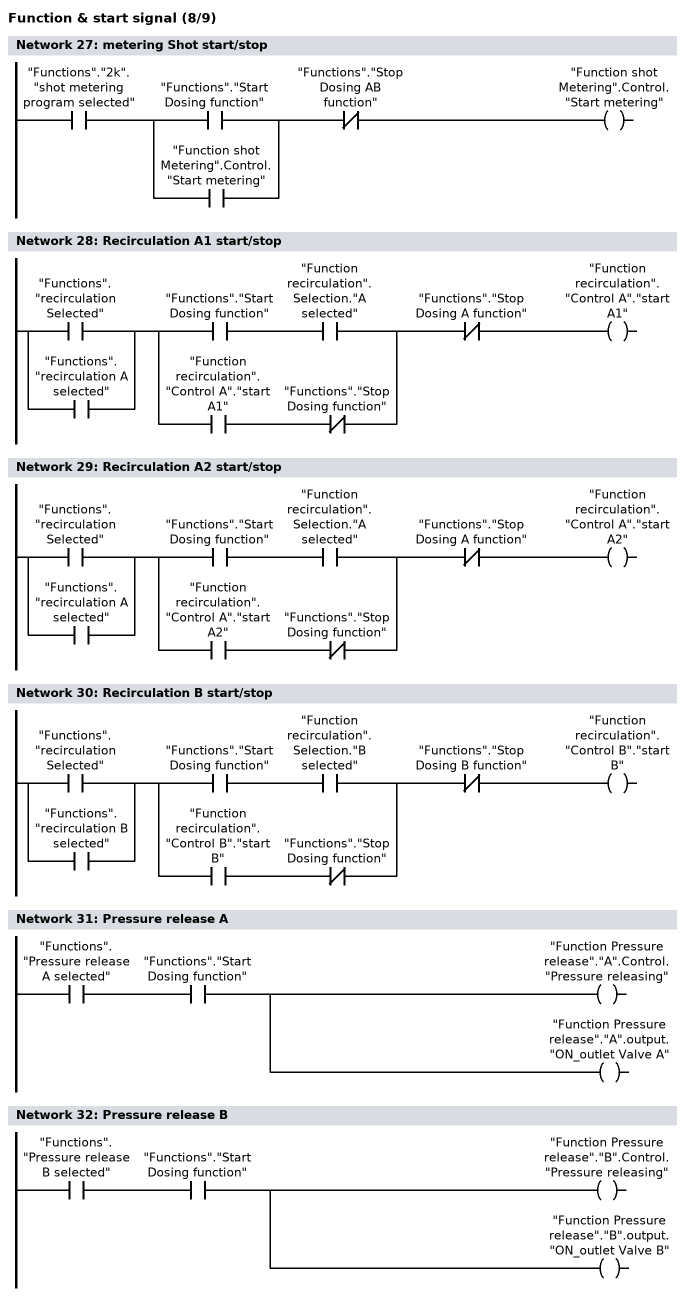
   RUNG wire#powerrail
      Contact( "Functions"."2k"."shot metering program selected" )
      wire#w1
      Contact( "Functions"."Start Dosing function" )
      wire#w2
      I_Contact( "Functions"."Stop Dosing AB function" )
      Coil( "Function shot Metering".Control."Start metering" )
   END_RUNG
   RUNG wire#w1
      Contact( "Function shot Metering".Control."Start metering" )
   END_RUNG wire#w2
   // the same network as SCL:
   "Function shot Metering".Control."Start metering" := "Functions"."2k"."shot metering program selected" AND ("Functions"."Start Dosing function" OR "Function shot Metering".Control."Start metering") AND NOT "Functions"."Stop Dosing AB function";
END_REGION

REGION Network 28: Recirculation A1 start/stop
   RUNG wire#powerrail
      Contact( "Functions"."recirculation Selected" )
      wire#w1
      Contact( "Functions"."Start Dosing function" )
      Contact( "Function recirculation".Selection."A selected" )
      wire#w2
      I_Contact( "Functions"."Stop Dosing A function" )
      Coil( "Function recirculation"."Control A"."start A1" )
   END_RUNG
   RUNG wire#powerrail
      Contact( "Functions"."recirculation A selected" )
   END_RUNG wire#w1
   RUNG wire#w1
      Contact( "Function recirculation"."Control A"."start A1" )
      I_Contact( "Functions"."Stop Dosing function" )
   END_RUNG wire#w2
   // the same network as SCL:
   "Function recirculation"."Control A"."start A1" := ("Functions"."recirculation Selected" OR "Functions"."recirculation A selected") AND (("Functions"."Start Dosing function" AND "Function recirculation".Selection."A selected") OR ("Function recirculation"."Control A"."start A1" AND NOT "Functions"."Stop Dosing function")) AND NOT "Functions"."Stop Dosing A function";
END_REGION

REGION Network 29: Recirculation A2 start/stop
   RUNG wire#powerrail
      Contact( "Functions"."recirculation Selected" )
      wire#w1
      Contact( "Functions"."Start Dosing function" )
      Contact( "Function recirculation".Selection."A selected" )
      wire#w2
      I_Contact( "Functions"."Stop Dosing A function" )
      Coil( "Function recirculation"."Control A"."start A2" )
   END_RUNG
   RUNG wire#powerrail
      Contact( "Functions"."recirculation A selected" )
   END_RUNG wire#w1
   RUNG wire#w1
      Contact( "Function recirculation"."Control A"."start A2" )
      I_Contact( "Functions"."Stop Dosing function" )
   END_RUNG wire#w2
   // the same network as SCL:
   "Function recirculation"."Control A"."start A2" := ("Functions"."recirculation Selected" OR "Functions"."recirculation A selected") AND (("Functions"."Start Dosing function" AND "Function recirculation".Selection."A selected") OR ("Function recirculation"."Control A"."start A2" AND NOT "Functions"."Stop Dosing function")) AND NOT "Functions"."Stop Dosing A function";
END_REGION

REGION Network 30: Recirculation B start/stop
   RUNG wire#powerrail
      Contact( "Functions"."recirculation Selected" )
      wire#w1
      Contact( "Functions"."Start Dosing function" )
      Contact( "Function recirculation".Selection."B selected" )
      wire#w2
      I_Contact( "Functions"."Stop Dosing B function" )
      Coil( "Function recirculation"."Control B"."start B" )
   END_RUNG
   RUNG wire#powerrail
      Contact( "Functions"."recirculation B selected" )
   END_RUNG wire#w1
   RUNG wire#w1
      Contact( "Function recirculation"."Control B"."start B" )
      I_Contact( "Functions"."Stop Dosing function" )
   END_RUNG wire#w2
   // the same network as SCL:
   "Function recirculation"."Control B"."start B" := ("Functions"."recirculation Selected" OR "Functions"."recirculation B selected") AND (("Functions"."Start Dosing function" AND "Function recirculation".Selection."B selected") OR ("Function recirculation"."Control B"."start B" AND NOT "Functions"."Stop Dosing function")) AND NOT "Functions"."Stop Dosing B function";
END_REGION

REGION Network 31: Pressure release A
   RUNG wire#powerrail
      Contact( "Functions"."Pressure release A selected" )
      Contact( "Functions"."Start Dosing function" )
      wire#w1
      Coil( "Function Pressure release"."A".Control."Pressure releasing" )
   END_RUNG
   RUNG wire#w1
      Coil( "Function Pressure release"."A".output."ON_outlet Valve A" )
   END_RUNG
   // the same network as SCL:
   "Function Pressure release"."A".Control."Pressure releasing" := "Functions"."Pressure release A selected" AND "Functions"."Start Dosing function";
   "Function Pressure release"."A".output."ON_outlet Valve A" := "Function Pressure release"."A".Control."Pressure releasing";
END_REGION

REGION Network 32: Pressure release B
   RUNG wire#powerrail
      Contact( "Functions"."Pressure release B selected" )
      Contact( "Functions"."Start Dosing function" )
      wire#w1
      Coil( "Function Pressure release"."B".Control."Pressure releasing" )
   END_RUNG
   RUNG wire#w1
      Coil( "Function Pressure release"."B".output."ON_outlet Valve B" )
   END_RUNG
   // the same network as SCL:
   "Function Pressure release"."B".Control."Pressure releasing" := "Functions"."Pressure release B selected" AND "Functions"."Start Dosing function";
   "Function Pressure release"."B".output."ON_outlet Valve B" := "Function Pressure release"."B".Control."Pressure releasing";
END_REGION

REGION Network 33: Pressure release AB
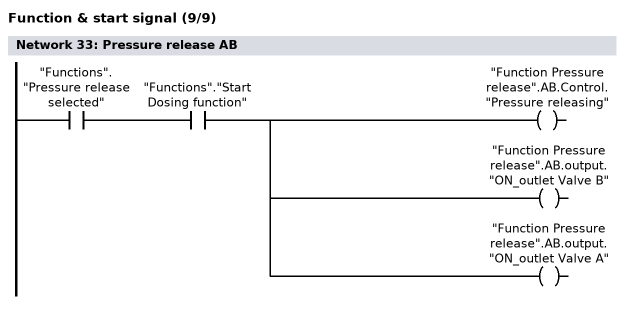
   RUNG wire#powerrail
      Contact( "Functions"."Pressure release selected" )
      Contact( "Functions"."Start Dosing function" )
      wire#w1
      Coil( "Function Pressure release".AB.Control."Pressure releasing" )
   END_RUNG
   RUNG wire#w1
      Coil( "Function Pressure release".AB.output."ON_outlet Valve B" )
   END_RUNG
   RUNG wire#w1
      Coil( "Function Pressure release".AB.output."ON_outlet Valve A" )
   END_RUNG
   // the same network as SCL:
   "Function Pressure release".AB.Control."Pressure releasing" := "Functions"."Pressure release selected" AND "Functions"."Start Dosing function";
   "Function Pressure release".AB.output."ON_outlet Valve B" := "Function Pressure release".AB.Control."Pressure releasing";
   "Function Pressure release".AB.output."ON_outlet Valve A" := "Function Pressure release".AB.Control."Pressure releasing";
END_REGION
END_FUNCTION

FUNCTION "Metering Program sequences" : Void   // FC2, LAD
{ S7_Optimized_Access := 'TRUE' }
VERSION : 0.1
// stored: AutoNumber true, IsIECCheckEnabled false, SetENOAutomatically false, UDAEnableTagReadback false
   VAR_TEMP
      temp1 : Bool;
   END_VAR
   VAR_TEMP   // added for the SCL form of the ladder/FBD networks
      _w1 : Bool;
   END_VAR
BEGIN

REGION Network 1: Do continous metering selection
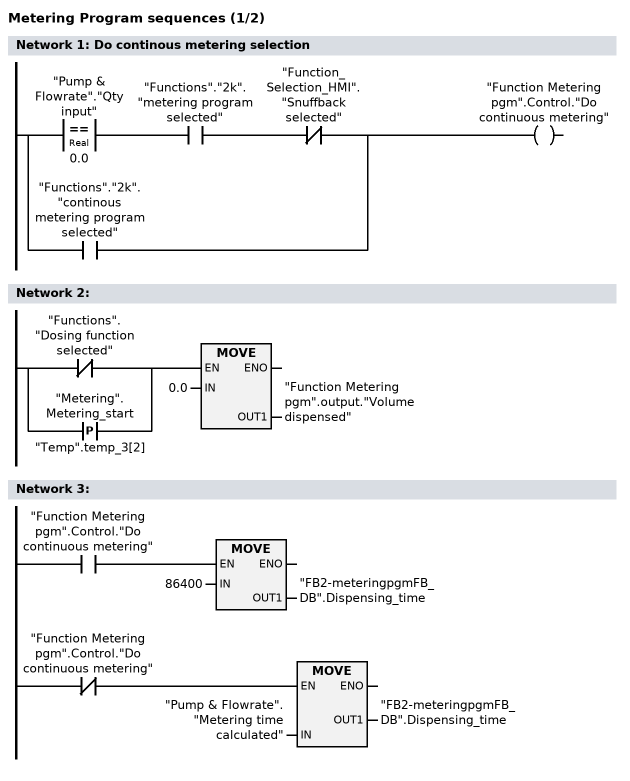
   RUNG wire#powerrail
      { S7_Templates := "SrcType := Real" } EQ_Contact(in1 := "Pump & Flowrate"."Qty input", in2 := 0.0)
      Contact( "Functions"."2k"."metering program selected" )
      I_Contact( "Function_Selection_HMI"."Snuffback selected" )
      wire#w1
      Coil( "Function Metering pgm".Control."Do continuous metering" )
   END_RUNG
   RUNG wire#powerrail
      Contact( "Functions"."2k"."continous metering program selected" )
   END_RUNG wire#w1
   // the same network as SCL:
   "Function Metering pgm".Control."Do continuous metering" := (("Pump & Flowrate"."Qty input" = 0.0) AND "Functions"."2k"."metering program selected" AND NOT "Function_Selection_HMI"."Snuffback selected") OR "Functions"."2k"."continous metering program selected";
END_REGION

REGION Network 2
   RUNG wire#powerrail
      I_Contact( "Functions"."Dosing function selected" )
      wire#w1
      Move(in := 0.0, out1 => "Function Metering pgm".output."Volume dispensed")
   END_RUNG
   RUNG wire#powerrail
      P_Contact(operand := "Metering".Metering_start, bit := "Temp".temp_3[2])
   END_RUNG wire#w1
   // the same network as SCL:
   #_w1 := "Metering".Metering_start AND NOT "Temp".temp_3[2];   // rising edge of "Metering".Metering_start
   "Temp".temp_3[2] := "Metering".Metering_start;
   IF NOT "Functions"."Dosing function selected" OR #_w1 THEN
       "Function Metering pgm".output."Volume dispensed" := 0.0;
   END_IF;
END_REGION

REGION Network 3
   RUNG wire#powerrail
      Contact( "Function Metering pgm".Control."Do continuous metering" )
      Move(in := 86400, out1 => "FB2-meteringpgmFB_DB".Dispensing_time)
   END_RUNG
   RUNG wire#powerrail
      I_Contact( "Function Metering pgm".Control."Do continuous metering" )
      Move(in := "Pump & Flowrate"."Metering time calculated", out1 => "FB2-meteringpgmFB_DB".Dispensing_time)
   END_RUNG
   // the same network as SCL:
   IF "Function Metering pgm".Control."Do continuous metering" THEN
       "FB2-meteringpgmFB_DB".Dispensing_time := 86400;
   END_IF;
   IF NOT "Function Metering pgm".Control."Do continuous metering" THEN
       "FB2-meteringpgmFB_DB".Dispensing_time := "Pump & Flowrate"."Metering time calculated";
   END_IF;
END_REGION

REGION Network 4
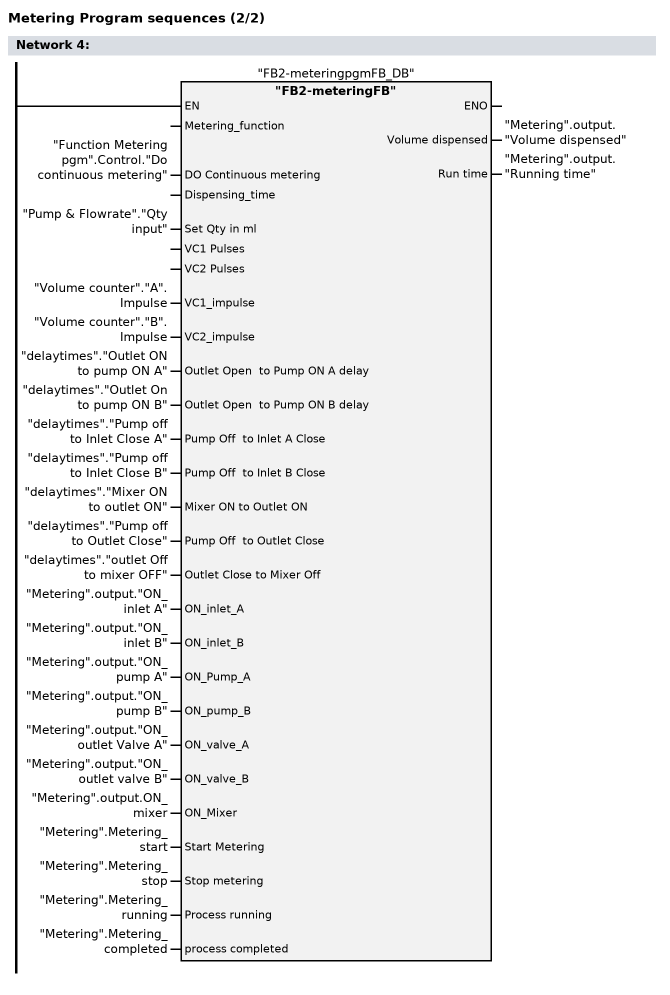
   RUNG wire#powerrail
      "FB2-meteringpgmFB_DB"(Metering_function :=, "DO Continuous metering" := "Function Metering pgm".Control."Do continuous metering", Dispensing_time :=, "Set Qty in ml" := "Pump & Flowrate"."Qty input", "VC1 Pulses" :=, "VC2 Pulses" :=, VC1_impulse := "Volume counter"."A".Impulse, VC2_impulse := "Volume counter"."B".Impulse, "Outlet Open  to Pump ON A delay" := "delaytimes"."Outlet ON to pump ON A", "Outlet Open  to Pump ON B delay" := "delaytimes"."Outlet On to pump ON B", "Pump Off  to Inlet A Close" := "delaytimes"."Pump off to Inlet Close A", "Pump Off  to Inlet B Close" := "delaytimes"."Pump off to Inlet Close B", "Mixer ON to Outlet ON" := "delaytimes"."Mixer ON to outlet ON", "Pump Off  to Outlet Close" := "delaytimes"."Pump off to Outlet Close", "Outlet Close to Mixer Off" := "delaytimes"."outlet Off to mixer OFF", ON_inlet_A := "Metering".output."ON_inlet A", ON_inlet_B := "Metering".output."ON_inlet B", ON_Pump_A := "Metering".output."ON_pump A", ON_pump_B := "Metering".output."ON_pump B", ON_valve_A := "Metering".output."ON_outlet Valve A", ON_valve_B := "Metering".output."ON_outlet valve B", ON_Mixer := "Metering".output.ON_mixer, "Start Metering" := "Metering".Metering_start, "Stop metering" := "Metering".Metering_stop, "Process running" := "Metering".Metering_running, "process completed" := "Metering".Metering_completed, "Volume dispensed" => "Metering".output."Volume dispensed", "Run time" => "Metering".output."Running time")
   END_RUNG
   // the same network as SCL:
   "FB2-meteringpgmFB_DB"("DO Continuous metering" := "Function Metering pgm".Control."Do continuous metering",   // "FB2-meteringFB"
                          "Set Qty in ml" := "Pump & Flowrate"."Qty input",
                          VC1_impulse := "Volume counter"."A".Impulse,
                          VC2_impulse := "Volume counter"."B".Impulse,
                          "Outlet Open  to Pump ON A delay" := "delaytimes"."Outlet ON to pump ON A",
                          "Outlet Open  to Pump ON B delay" := "delaytimes"."Outlet On to pump ON B",
                          "Pump Off  to Inlet A Close" := "delaytimes"."Pump off to Inlet Close A",
                          "Pump Off  to Inlet B Close" := "delaytimes"."Pump off to Inlet Close B",
                          "Mixer ON to Outlet ON" := "delaytimes"."Mixer ON to outlet ON",
                          "Pump Off  to Outlet Close" := "delaytimes"."Pump off to Outlet Close",
                          "Outlet Close to Mixer Off" := "delaytimes"."outlet Off to mixer OFF",
                          ON_inlet_A := "Metering".output."ON_inlet A",
                          ON_inlet_B := "Metering".output."ON_inlet B",
                          ON_Pump_A := "Metering".output."ON_pump A",
                          ON_pump_B := "Metering".output."ON_pump B",
                          ON_valve_A := "Metering".output."ON_outlet Valve A",
                          ON_valve_B := "Metering".output."ON_outlet valve B",
                          ON_Mixer := "Metering".output.ON_mixer,
                          "Start Metering" := "Metering".Metering_start,
                          "Stop metering" := "Metering".Metering_stop,
                          "Process running" := "Metering".Metering_running,
                          "process completed" := "Metering".Metering_completed,
                          "Volume dispensed" => "Metering".output."Volume dispensed",
                          "Run time" => "Metering".output."Running time");
END_REGION

REGION Network 5 (SCL)
   //IF NOT ("Gear Pump B On_REW") AND NOT ("Gear Pump A On_REW") THEN
       IF "Functions"."2k"."continous metering program selected" THEN
           "Function Continous Metering pgm".output."Volume dispensed" := "Metering".output."Volume dispensed";
           "Function Continous Metering pgm".output."Running time" := "Metering".output."Running time";
       ELSIF "Functions"."2k"."metering program selected" THEN
           "Function Metering pgm".output."Volume dispensed" := "Metering".output."Volume dispensed";
           "Function Metering pgm".output."Running time" := "Metering".output."Running time";
       ELSIF "Functions"."2k"."shot metering program selected" THEN
           "Function shot Metering".output."Volume dispensed" := "Metering".output."Volume dispensed";
           "Function shot Metering".output."Running time" := "Metering".output."Running time";
       ELSIF "Functions"."2k"."pre run program selected" THEN
           "Function Pre run".output."Volume dispensed" := "Metering".output."Volume dispensed";
           "Function Pre run".output."Running time" := "Metering".output."Running time";
       END_IF;
   //END_IF;
END_REGION

REGION Network 6 (SCL): Prerun Completed
   IF "Functions"."2k"."pre run program selected" AND "Metering".Metering_completed THEN //AND  ("Function Pre run".output."Volume dispensed" >="Pump & Flowrate"."Qty input")
       "Function Pre run".Control."metering completed" := TRUE;
   ELSIF "Function Flush"."Control A"."flush running" OR "Function Dearing with valve"."Control A"."dearing running"
       OR "Function Dearing with valve"."Control B"."dearing running" OR "Potlife".contol."Potlife elapsed machine not in regeneration"
           THEN //OR ("Functions"."2k"."pre run program selected"  AND "Functions"."Stop Dosing function")

       "Function Pre run".Control."metering completed" := FALSE;
   END_IF;
   "Control"."waiting For pre run" := NOT ("Function Pre run".Control."metering completed");
END_REGION
END_FUNCTION

FUNCTION_BLOCK "FB2-meteringFB"   // FB2, LAD
{ S7_Optimized_Access := 'TRUE' }
VERSION : 0.1
// stored: AutoNumber true, IsIECCheckEnabled false, IsRetainMemResEnabled false, MemoryReserve 100, SetENOAutomatically false, UDAEnableTagReadback false
   VAR_INPUT
      Metering_function : Int;
      "DO Continuous metering" : Bool;
      Dispensing_time : DInt;
      "Set Qty in ml" : Real;
      "VC1 Pulses" : DInt;
      "VC2 Pulses" : DInt;
      VC1_impulse : Real;
      VC2_impulse : Real;
      "Outlet Open  to Pump ON A delay" : DInt;
      "Outlet Open  to Pump ON B delay" : DInt;
      "Pump Off  to Inlet A Close" : DInt;
      "Pump Off  to Inlet B Close" : DInt;
      "Mixer ON to Outlet ON" : DInt;
      "Pump Off  to Outlet Close" : DInt;
      "Outlet Close to Mixer Off" : DInt;
   END_VAR
   VAR_OUTPUT
      "Volume dispensed" : Real;
      "Run time" : Int;
   END_VAR
   VAR_IN_OUT
      ON_inlet_A : Bool;
      ON_inlet_B : Bool;
      ON_Pump_A : Bool;
      ON_pump_B : Bool;
      ON_valve_A : Bool;
      ON_valve_B : Bool;
      ON_Mixer : Bool;
      "Start Metering" : Bool;
      "Stop metering" : Bool;
      "Process running" : Bool;
      "process completed" : Bool;
   END_VAR
   VAR
      "pump A to valveA delay" : Bool;
      "Pump B to valve B delay" : Bool;
      "Pump Off to mixer off delay_1" : Bool;
      "VC1 pulses prev" : DInt;
      "VC2 pulses prev" : DInt;
      "VC1 pulse generted" : DInt;
      "VC2 pulse generated" : DInt;
      "Pump A Voulme dispensed" : Real;
      "Pump B volume dispensed" : Real;
      "Total Volume dispensed" : Real;
      "metering started" : Bool;
      "metering time in msec" : DInt;
      "dispense time elapsed" : Bool;
      R_TRIG_Instance { S7_SetPoint := 'True'} : R_TRIG;
      IEC_Timer_0_Instance { S7_SetPoint := 'True'} : TON_TIME;
      IEC_Timer_0_Instance_1 { S7_SetPoint := 'True'} : TON_TIME;
      IEC_Timer_0_Instance_2 { S7_SetPoint := 'True'} : TON_TIME;
      R_TRIG_Instance_1 { S7_SetPoint := 'True'} : R_TRIG;
      temp { S7_SetPoint := 'True'} : Bool;
      IEC_Timer_0_Instance_3 { S7_SetPoint := 'True'} : TON_TIME;
      IEC_Timer_0_Instance_4 { S7_SetPoint := 'True'} : TON_TIME;
      IEC_Timer_0_Instance_5 { S7_SetPoint := 'True'} : TON_TIME;
      IEC_Timer_0_Instance_6 { S7_SetPoint := 'True'} : TON_TIME;
      IEC_Timer_0_Instance_7 { S7_SetPoint := 'True'} : TON_TIME;
      IEC_Timer_0_Instance_8 { S7_SetPoint := 'True'} : TON_TIME;
   END_VAR
   VAR_TEMP
      Ons_temp : Bool;
   END_VAR
   VAR_TEMP   // added for the SCL form of the ladder/FBD networks
      _w1 : Bool;
      _w2 : Bool;
      _w3 : Bool;
   END_VAR
BEGIN

REGION Network 1
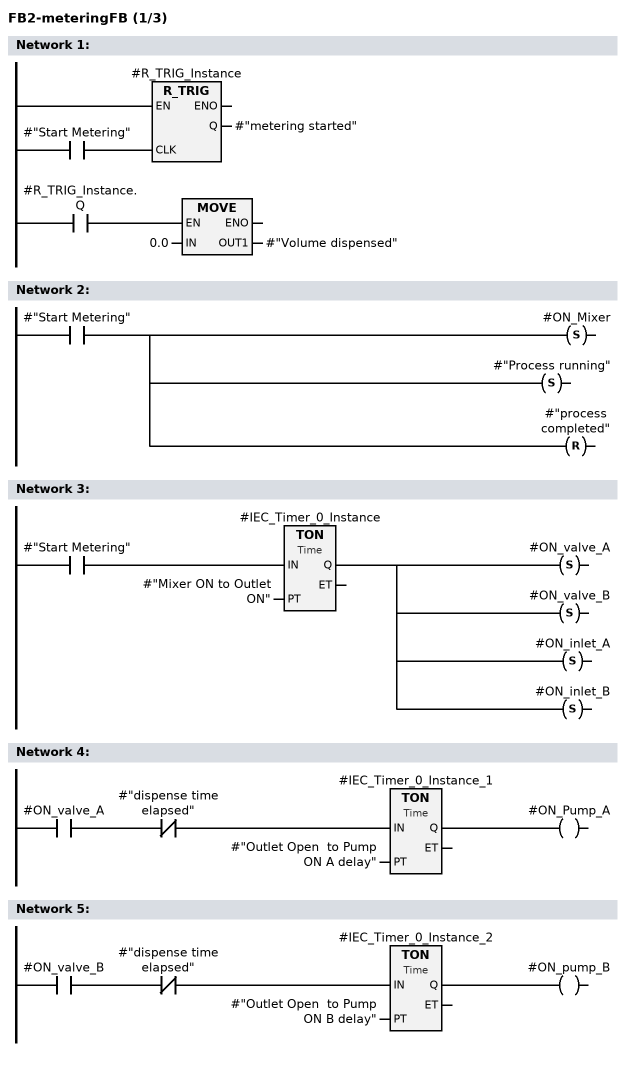
   RUNG wire#powerrail
      #R_TRIG_Instance.R_TRIG(CLK := wire#w1, Q => #"metering started")
   END_RUNG
   RUNG wire#powerrail
      Contact( #"Start Metering" )
   END_RUNG wire#w1
   RUNG wire#powerrail
      Contact( #R_TRIG_Instance.Q )
      Move(in := 0.0, out1 => #"Volume dispensed")
   END_RUNG
   // the same network as SCL:
   #R_TRIG_Instance(CLK := #"Start Metering", Q => #"metering started");   // R_TRIG
   IF #R_TRIG_Instance.Q THEN #"Volume dispensed" := 0.0; END_IF;
END_REGION

REGION Network 2
   RUNG wire#powerrail
      Contact( #"Start Metering" )
      wire#w1
      S_Coil( #ON_Mixer )
   END_RUNG
   RUNG wire#w1
      S_Coil( #"Process running" )
   END_RUNG
   RUNG wire#w1
      R_Coil( #"process completed" )
   END_RUNG
   // the same network as SCL:
   IF #"Start Metering" THEN
       #ON_Mixer := TRUE;
       #"Process running" := TRUE;
       #"process completed" := FALSE;
   END_IF;
END_REGION

REGION Network 3
   RUNG wire#powerrail
      Contact( #"Start Metering" )
      { S7_Templates := "time_type := Time" } #IEC_Timer_0_Instance.TON(pt := #"Mixer ON to Outlet ON", et =>)
      wire#w1
      S_Coil( #ON_valve_A )
   END_RUNG
   RUNG wire#w1
      S_Coil( #ON_valve_B )
   END_RUNG
   RUNG wire#w1
      S_Coil( #ON_inlet_A )
   END_RUNG
   RUNG wire#w1
      S_Coil( #ON_inlet_B )
   END_RUNG
   // the same network as SCL:
   #IEC_Timer_0_Instance(IN := #"Start Metering", PT := #"Mixer ON to Outlet ON");   // TON
   IF #IEC_Timer_0_Instance.Q THEN
       #ON_valve_A := TRUE;
       #ON_valve_B := TRUE;
       #ON_inlet_A := TRUE;
       #ON_inlet_B := TRUE;
   END_IF;
END_REGION

REGION Network 4
   RUNG wire#powerrail
      Contact( #ON_valve_A )
      I_Contact( #"dispense time elapsed" )
      { S7_Templates := "time_type := Time" } #IEC_Timer_0_Instance_1.TON(pt := #"Outlet Open  to Pump ON A delay", et =>)
      Coil( #ON_Pump_A )
   END_RUNG
   // the same network as SCL:
   #IEC_Timer_0_Instance_1(IN := #ON_valve_A AND NOT #"dispense time elapsed",   // TON
                           PT := #"Outlet Open  to Pump ON A delay");
   #ON_Pump_A := #IEC_Timer_0_Instance_1.Q;
END_REGION

REGION Network 5
   RUNG wire#powerrail
      Contact( #ON_valve_B )
      I_Contact( #"dispense time elapsed" )
      { S7_Templates := "time_type := Time" } #IEC_Timer_0_Instance_2.TON(pt := #"Outlet Open  to Pump ON B delay", et =>)
      Coil( #ON_pump_B )
   END_RUNG
   // the same network as SCL:
   #IEC_Timer_0_Instance_2(IN := #ON_valve_B AND NOT #"dispense time elapsed",   // TON
                           PT := #"Outlet Open  to Pump ON B delay");
   #ON_pump_B := #IEC_Timer_0_Instance_2.Q;
END_REGION

REGION Network 6
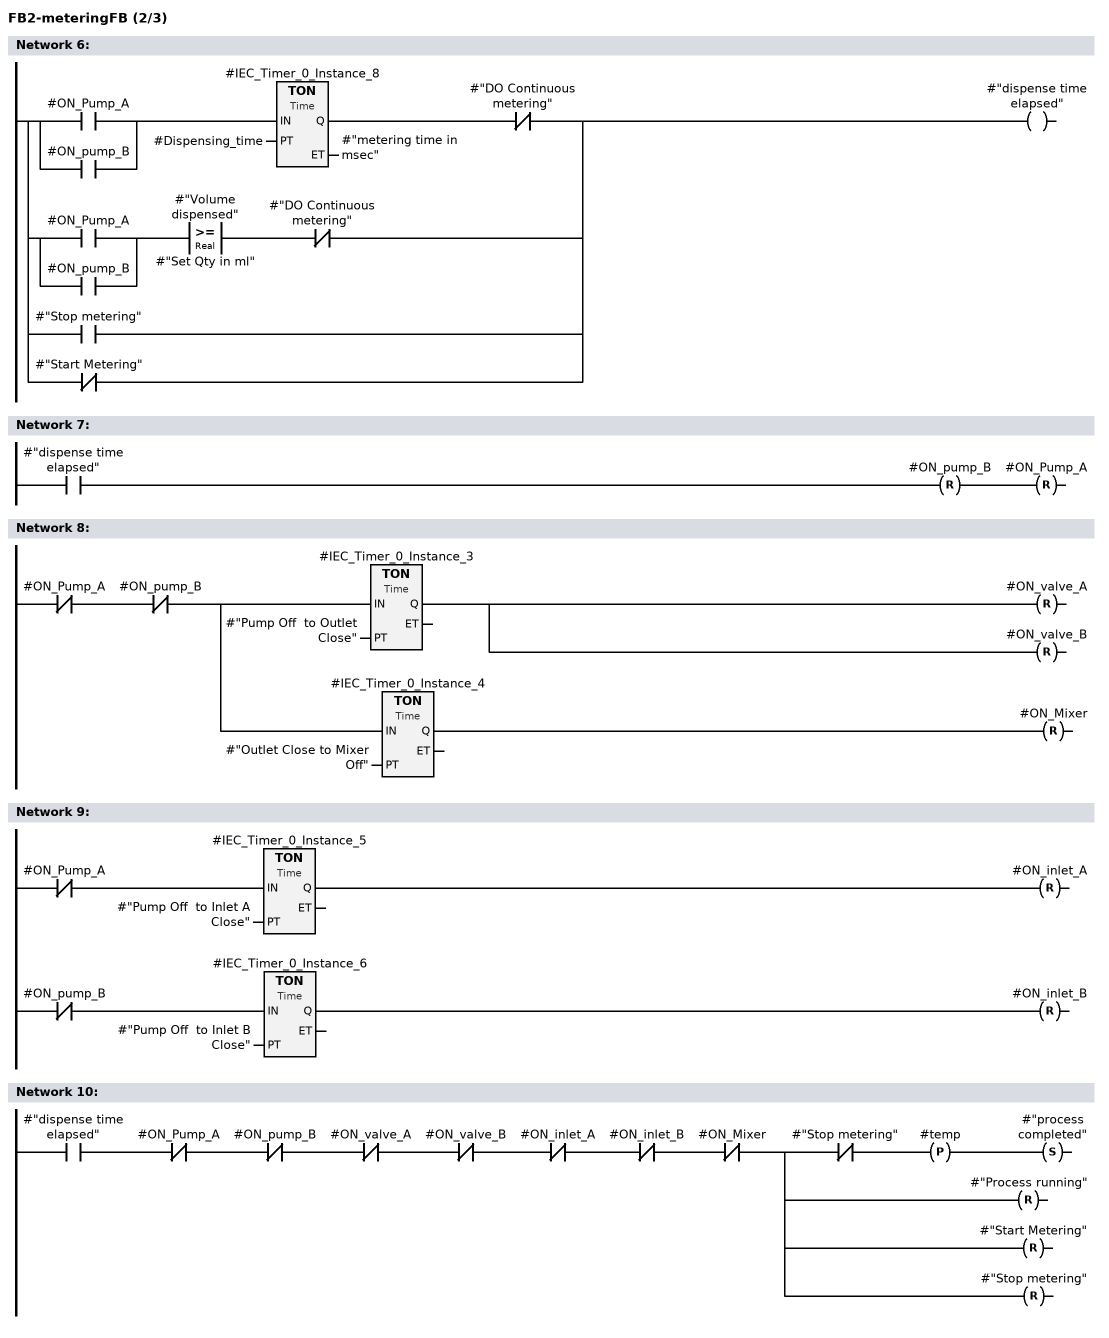
   RUNG wire#powerrail
      Contact( #ON_Pump_A )
      wire#w1
      { S7_Templates := "time_type := Time" } #IEC_Timer_0_Instance_8.TON(pt := #Dispensing_time, et => #"metering time in msec")
      I_Contact( #"DO Continuous metering" )
      wire#w2
      Coil( #"dispense time elapsed" )
   END_RUNG
   RUNG wire#powerrail
      Contact( #ON_pump_B )
   END_RUNG wire#w1
   RUNG wire#powerrail
      Contact( #ON_Pump_A )
      wire#w3
      { S7_Templates := "SrcType := Real" } GE_Contact(in1 := #"Volume dispensed", in2 := #"Set Qty in ml")
      I_Contact( #"DO Continuous metering" )
   END_RUNG wire#w2
   RUNG wire#powerrail
      Contact( #ON_pump_B )
   END_RUNG wire#w3
   RUNG wire#powerrail
      Contact( #"Stop metering" )
   END_RUNG wire#w2
   RUNG wire#powerrail
      I_Contact( #"Start Metering" )
   END_RUNG wire#w2
   // the same network as SCL:
   #IEC_Timer_0_Instance_8(IN := #ON_Pump_A OR #ON_pump_B,   // TON
                           PT := #Dispensing_time,
                           ET => #"metering time in msec");
   #"dispense time elapsed" := (#IEC_Timer_0_Instance_8.Q AND NOT #"DO Continuous metering") OR ((#ON_Pump_A OR #ON_pump_B) AND (#"Volume dispensed" >= #"Set Qty in ml") AND NOT #"DO Continuous metering") OR #"Stop metering" OR NOT #"Start Metering";
END_REGION

REGION Network 7
   RUNG wire#powerrail
      Contact( #"dispense time elapsed" )
      R_Coil( #ON_pump_B )
      R_Coil( #ON_Pump_A )
   END_RUNG
   // the same network as SCL:
   IF #"dispense time elapsed" THEN
       #ON_pump_B := FALSE;
       #ON_Pump_A := FALSE;
   END_IF;
END_REGION

REGION Network 8
   RUNG wire#powerrail
      I_Contact( #ON_Pump_A )
      I_Contact( #ON_pump_B )
      wire#w1
      { S7_Templates := "time_type := Time" } #IEC_Timer_0_Instance_3.TON(pt := #"Pump Off  to Outlet Close", et =>)
      wire#w2
      R_Coil( #ON_valve_A )
   END_RUNG
   RUNG wire#w2
      R_Coil( #ON_valve_B )
   END_RUNG
   RUNG wire#w1
      { S7_Templates := "time_type := Time" } #IEC_Timer_0_Instance_4.TON(pt := #"Outlet Close to Mixer Off", et =>)
      R_Coil( #ON_Mixer )
   END_RUNG
   // the same network as SCL:
   #_w1 := NOT #ON_Pump_A AND NOT #ON_pump_B;
   #IEC_Timer_0_Instance_3(IN := #_w1, PT := #"Pump Off  to Outlet Close");   // TON
   IF #IEC_Timer_0_Instance_3.Q THEN
       #ON_valve_A := FALSE;
       #ON_valve_B := FALSE;
   END_IF;
   #IEC_Timer_0_Instance_4(IN := #_w1, PT := #"Outlet Close to Mixer Off");   // TON
   IF #IEC_Timer_0_Instance_4.Q THEN #ON_Mixer := FALSE; END_IF;
END_REGION

REGION Network 9
   RUNG wire#powerrail
      I_Contact( #ON_Pump_A )
      { S7_Templates := "time_type := Time" } #IEC_Timer_0_Instance_5.TON(pt := #"Pump Off  to Inlet A Close", et =>)
      R_Coil( #ON_inlet_A )
   END_RUNG
   RUNG wire#powerrail
      I_Contact( #ON_pump_B )
      { S7_Templates := "time_type := Time" } #IEC_Timer_0_Instance_6.TON(pt := #"Pump Off  to Inlet B Close", et =>)
      R_Coil( #ON_inlet_B )
   END_RUNG
   // the same network as SCL:
   #IEC_Timer_0_Instance_5(IN := NOT #ON_Pump_A, PT := #"Pump Off  to Inlet A Close");   // TON
   IF #IEC_Timer_0_Instance_5.Q THEN #ON_inlet_A := FALSE; END_IF;
   #IEC_Timer_0_Instance_6(IN := NOT #ON_pump_B, PT := #"Pump Off  to Inlet B Close");   // TON
   IF #IEC_Timer_0_Instance_6.Q THEN #ON_inlet_B := FALSE; END_IF;
END_REGION

REGION Network 10
   RUNG wire#powerrail
      Contact( #"dispense time elapsed" )
      I_Contact( #ON_Pump_A )
      I_Contact( #ON_pump_B )
      I_Contact( #ON_valve_A )
      I_Contact( #ON_valve_B )
      I_Contact( #ON_inlet_A )
      I_Contact( #ON_inlet_B )
      I_Contact( #ON_Mixer )
      wire#w1
      I_Contact( #"Stop metering" )
      P_Trig( #temp )
      S_Coil( #"process completed" )
   END_RUNG
   RUNG wire#w1
      R_Coil( #"Process running" )
   END_RUNG
   RUNG wire#w1
      R_Coil( #"Start Metering" )
   END_RUNG
   RUNG wire#w1
      R_Coil( #"Stop metering" )
   END_RUNG
   // the same network as SCL:
   #_w1 := #"dispense time elapsed" AND NOT #ON_Pump_A AND NOT #ON_pump_B AND NOT #ON_valve_A AND NOT #ON_valve_B AND NOT #ON_inlet_A AND NOT #ON_inlet_B AND NOT #ON_Mixer;
   #_w2 := #_w1 AND NOT #"Stop metering";
   #_w3 := #_w2 AND NOT #temp;   // rising edge
   #temp := #_w2;
   IF #_w3 THEN #"process completed" := TRUE; END_IF;
   IF #_w1 THEN
       #"Process running" := FALSE;
       #"Start Metering" := FALSE;
       #"Stop metering" := FALSE;
   END_IF;
END_REGION

REGION Network 11
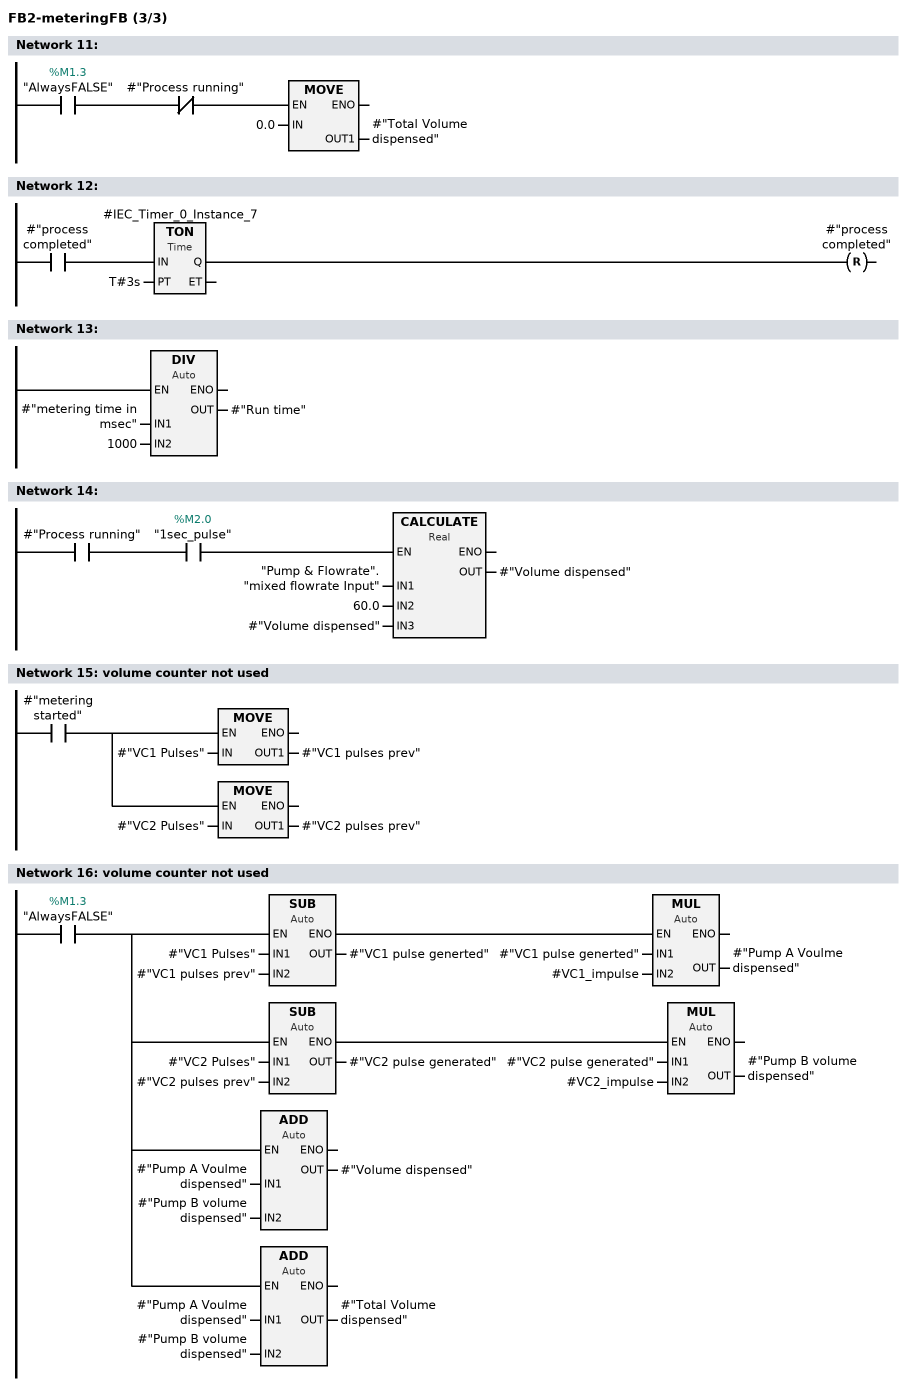
   RUNG wire#powerrail
      Contact( "AlwaysFALSE" )
      I_Contact( #"Process running" )
      Move(in := 0.0, out1 => #"Total Volume dispensed")
   END_RUNG
   // the same network as SCL:
   IF "AlwaysFALSE" AND NOT #"Process running" THEN #"Total Volume dispensed" := 0.0; END_IF;
END_REGION

REGION Network 12
   RUNG wire#powerrail
      Contact( #"process completed" )
      { S7_Templates := "time_type := Time" } #IEC_Timer_0_Instance_7.TON(pt := T#3s, et =>)
      R_Coil( #"process completed" )
   END_RUNG
   // the same network as SCL:
   #IEC_Timer_0_Instance_7(IN := #"process completed", PT := T#3s);   // TON
   IF #IEC_Timer_0_Instance_7.Q THEN #"process completed" := FALSE; END_IF;
END_REGION

REGION Network 13
   RUNG wire#powerrail
      Div(in1 := #"metering time in msec", in2 := 1000, out => #"Run time")
   END_RUNG
   // the same network as SCL:
   #"Run time" := #"metering time in msec" / 1000;
END_REGION

REGION Network 14
   RUNG wire#powerrail
      Contact( #"Process running" )
      Contact( "1sec_pulse" )
      { S7_Templates := "SrcType := Real"; S7_Expression := "(IN1/IN2)+IN3" } Calculate(in1 := "Pump & Flowrate"."mixed flowrate Input", in2 := 60.0, in3 := #"Volume dispensed", out => #"Volume dispensed")
   END_RUNG
   // the same network as SCL:
   IF #"Process running" AND "1sec_pulse" THEN
       #"Volume dispensed" := ("Pump & Flowrate"."mixed flowrate Input"/60.0)+#"Volume dispensed";
   END_IF;
END_REGION

REGION Network 15: volume counter not used
   RUNG wire#powerrail
      Contact( #"metering started" )
      wire#w1
      Move(in := #"VC1 Pulses", out1 => #"VC1 pulses prev")
   END_RUNG
   RUNG wire#w1
      Move(in := #"VC2 Pulses", out1 => #"VC2 pulses prev")
   END_RUNG
   // the same network as SCL:
   IF #"metering started" THEN
       #"VC1 pulses prev" := #"VC1 Pulses";
       #"VC2 pulses prev" := #"VC2 Pulses";
   END_IF;
END_REGION

REGION Network 16: volume counter not used
   RUNG wire#powerrail
      Contact( "AlwaysFALSE" )
      wire#w1
      Sub(in1 := #"VC1 Pulses", in2 := #"VC1 pulses prev", out => #"VC1 pulse generted")
      Mul(in1 := #"VC1 pulse generted", in2 := #VC1_impulse, out => #"Pump A Voulme dispensed")
   END_RUNG
   RUNG wire#w1
      Sub(in1 := #"VC2 Pulses", in2 := #"VC2 pulses prev", out => #"VC2 pulse generated")
      Mul(in1 := #"VC2 pulse generated", in2 := #VC2_impulse, out => #"Pump B volume dispensed")
   END_RUNG
   RUNG wire#w1
      Add(in1 := #"Pump A Voulme dispensed", in2 := #"Pump B volume dispensed", out => #"Volume dispensed")
   END_RUNG
   RUNG wire#w1
      Add(in1 := #"Pump A Voulme dispensed", in2 := #"Pump B volume dispensed", out => #"Total Volume dispensed")
   END_RUNG
   // the same network as SCL:
   IF "AlwaysFALSE" THEN
       #"VC1 pulse generted" := #"VC1 Pulses" - #"VC1 pulses prev";
       #"Pump A Voulme dispensed" := #"VC1 pulse generted" * #VC1_impulse;
       #"VC2 pulse generated" := #"VC2 Pulses" - #"VC2 pulses prev";
       #"Pump B volume dispensed" := #"VC2 pulse generated" * #VC2_impulse;
       #"Volume dispensed" := #"Pump A Voulme dispensed" + #"Pump B volume dispensed";
       #"Total Volume dispensed" := #"Pump A Voulme dispensed" + #"Pump B volume dispensed";
   END_IF;
END_REGION
END_FUNCTION_BLOCK

FUNCTION "Ratio Check Program sequences" : Void   // FC6, LAD
{ S7_Optimized_Access := 'TRUE' }
VERSION : 0.1
// stored: AutoNumber true, IsIECCheckEnabled false, SetENOAutomatically false, UDAEnableTagReadback false
   VAR_TEMP
      temp1 : Bool;
   END_VAR
   VAR_TEMP   // added for the SCL form of the ladder/FBD networks
      _w1 : Bool;
      _w2 : Bool;
      _w3 : Bool;
      _w4 : Bool;
   END_VAR
BEGIN

REGION Network 1
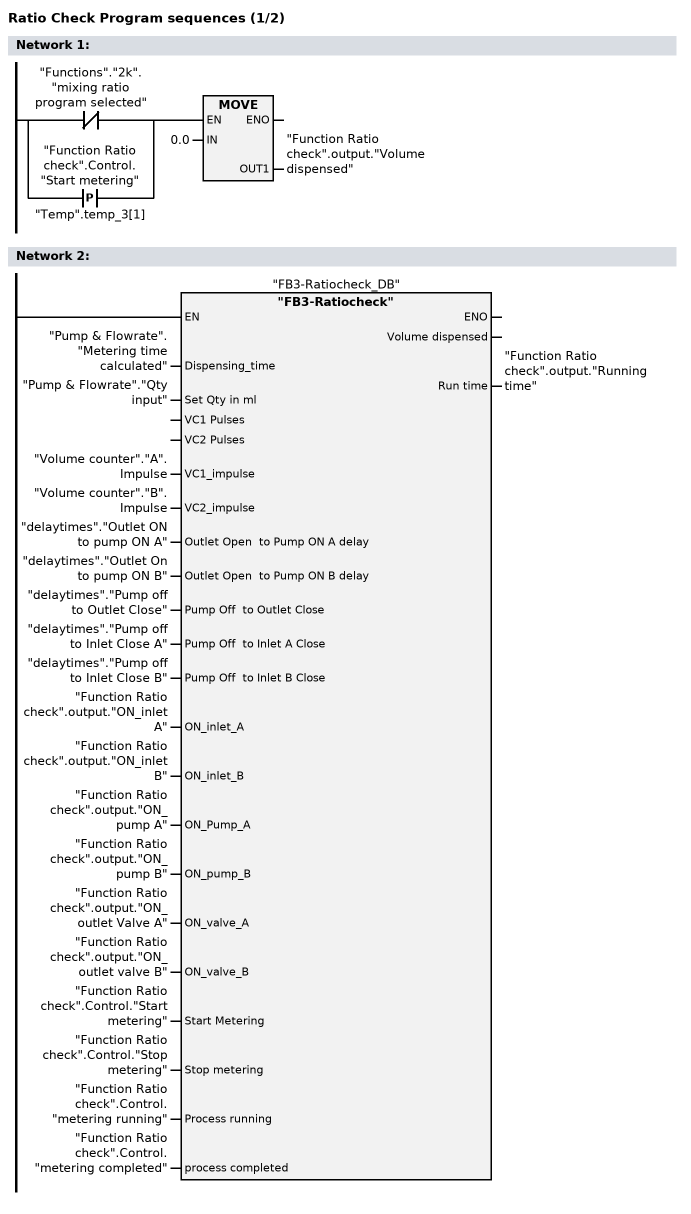
   RUNG wire#powerrail
      I_Contact( "Functions"."2k"."mixing ratio program selected" )
      wire#w1
      Move(in := 0.0, out1 => "Function Ratio check".output."Volume dispensed")
   END_RUNG
   RUNG wire#powerrail
      P_Contact(operand := "Function Ratio check".Control."Start metering", bit := "Temp".temp_3[1])
   END_RUNG wire#w1
   // the same network as SCL:
   #_w1 := "Function Ratio check".Control."Start metering" AND NOT "Temp".temp_3[1];   // rising edge of "Function Ratio check".Control."Start metering"
   "Temp".temp_3[1] := "Function Ratio check".Control."Start metering";
   IF NOT "Functions"."2k"."mixing ratio program selected" OR #_w1 THEN
       "Function Ratio check".output."Volume dispensed" := 0.0;
   END_IF;
END_REGION

REGION Network 2
   RUNG wire#powerrail
      "FB3-Ratiocheck_DB"(Dispensing_time := "Pump & Flowrate"."Metering time calculated", "Set Qty in ml" := "Pump & Flowrate"."Qty input", "VC1 Pulses" :=, "VC2 Pulses" :=, VC1_impulse := "Volume counter"."A".Impulse, VC2_impulse := "Volume counter"."B".Impulse, "Outlet Open  to Pump ON A delay" := "delaytimes"."Outlet ON to pump ON A", "Outlet Open  to Pump ON B delay" := "delaytimes"."Outlet On to pump ON B", "Pump Off  to Outlet Close" := "delaytimes"."Pump off to Outlet Close", "Pump Off  to Inlet A Close" := "delaytimes"."Pump off to Inlet Close A", "Pump Off  to Inlet B Close" := "delaytimes"."Pump off to Inlet Close B", ON_inlet_A := "Function Ratio check".output."ON_inlet A", ON_inlet_B := "Function Ratio check".output."ON_inlet B", ON_Pump_A := "Function Ratio check".output."ON_pump A", ON_pump_B := "Function Ratio check".output."ON_pump B", ON_valve_A := "Function Ratio check".output."ON_outlet Valve A", ON_valve_B := "Function Ratio check".output."ON_outlet valve B", "Start Metering" := "Function Ratio check".Control."Start metering", "Stop metering" := "Function Ratio check".Control."Stop metering", "Process running" := "Function Ratio check".Control."metering running", "process completed" := "Function Ratio check".Control."metering completed", "Volume dispensed" =>, "Run time" => "Function Ratio check".output."Running time")
   END_RUNG
   // the same network as SCL:
   "FB3-Ratiocheck_DB"(Dispensing_time := "Pump & Flowrate"."Metering time calculated",   // "FB3-Ratiocheck"
                       "Set Qty in ml" := "Pump & Flowrate"."Qty input",
                       VC1_impulse := "Volume counter"."A".Impulse,
                       VC2_impulse := "Volume counter"."B".Impulse,
                       "Outlet Open  to Pump ON A delay" := "delaytimes"."Outlet ON to pump ON A",
                       "Outlet Open  to Pump ON B delay" := "delaytimes"."Outlet On to pump ON B",
                       "Pump Off  to Outlet Close" := "delaytimes"."Pump off to Outlet Close",
                       "Pump Off  to Inlet A Close" := "delaytimes"."Pump off to Inlet Close A",
                       "Pump Off  to Inlet B Close" := "delaytimes"."Pump off to Inlet Close B",
                       ON_inlet_A := "Function Ratio check".output."ON_inlet A",
                       ON_inlet_B := "Function Ratio check".output."ON_inlet B",
                       ON_Pump_A := "Function Ratio check".output."ON_pump A",
                       ON_pump_B := "Function Ratio check".output."ON_pump B",
                       ON_valve_A := "Function Ratio check".output."ON_outlet Valve A",
                       ON_valve_B := "Function Ratio check".output."ON_outlet valve B",
                       "Start Metering" := "Function Ratio check".Control."Start metering",
                       "Stop metering" := "Function Ratio check".Control."Stop metering",
                       "Process running" := "Function Ratio check".Control."metering running",
                       "process completed" := "Function Ratio check".Control."metering completed",
                       "Run time" => "Function Ratio check".output."Running time");
END_REGION

REGION Network 3: Volume dispensed
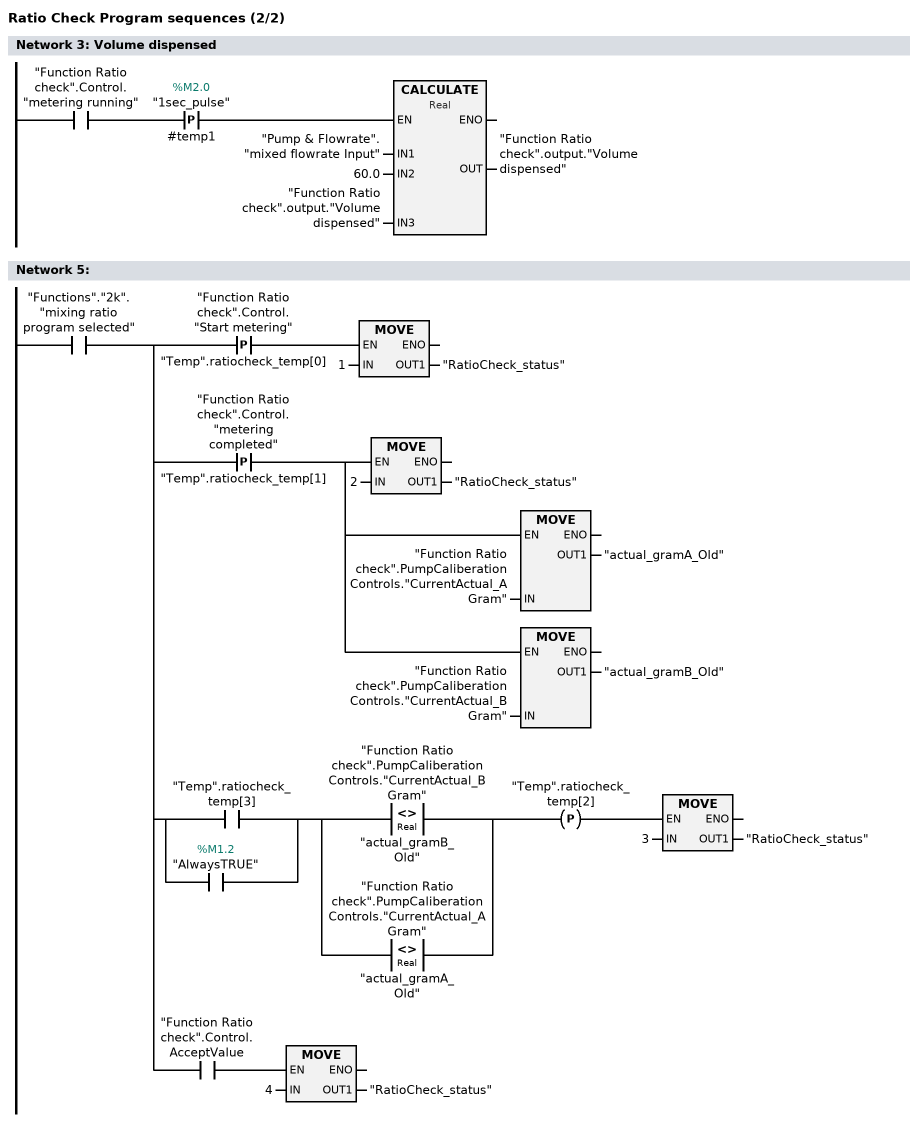
   RUNG wire#powerrail
      Contact( "Function Ratio check".Control."metering running" )
      P_Contact(operand := "1sec_pulse", bit := #temp1)
      { S7_Templates := "SrcType := Real"; S7_Expression := "(IN1/IN2)+IN3" } Calculate(in1 := "Pump & Flowrate"."mixed flowrate Input", in2 := 60.0, in3 := "Function Ratio check".output."Volume dispensed", out => "Function Ratio check".output."Volume dispensed")
   END_RUNG
   // the same network as SCL:
   #_w1 := "Function Ratio check".Control."metering running" AND "1sec_pulse" AND NOT #temp1;   // rising edge of "1sec_pulse"
   #temp1 := "1sec_pulse";
   IF #_w1 THEN
       "Function Ratio check".output."Volume dispensed" := ("Pump & Flowrate"."mixed flowrate Input"/60.0)+"Function Ratio check".output."Volume dispensed";
   END_IF;
END_REGION

REGION Network 5
   RUNG wire#powerrail
      Contact( "Functions"."2k"."mixing ratio program selected" )
      wire#w1
      P_Contact(operand := "Function Ratio check".Control."Start metering", bit := "Temp".ratiocheck_temp[0])
      Move(in := 1, out1 => "RatioCheck_status")
   END_RUNG
   RUNG wire#w1
      P_Contact(operand := "Function Ratio check".Control."metering completed", bit := "Temp".ratiocheck_temp[1])
      wire#w2
      Move(in := 2, out1 => "RatioCheck_status")
   END_RUNG
   RUNG wire#w2
      Move(in := "Function Ratio check".PumpCaliberationControls."CurrentActual_A Gram", out1 => "actual_gramA_Old")
   END_RUNG
   RUNG wire#w2
      Move(in := "Function Ratio check".PumpCaliberationControls."CurrentActual_B Gram", out1 => "actual_gramB_Old")
   END_RUNG
   RUNG wire#w1
      Contact( "Temp".ratiocheck_temp[3] )
      wire#w3
      { S7_Templates := "SrcType := Real" } NE_Contact(in1 := "Function Ratio check".PumpCaliberationControls."CurrentActual_B Gram", in2 := "actual_gramB_Old")
      wire#w4
      P_Trig( "Temp".ratiocheck_temp[2] )
      Move(in := 3, out1 => "RatioCheck_status")
   END_RUNG
   RUNG wire#w1
      Contact( "AlwaysTRUE" )
   END_RUNG wire#w3
   RUNG wire#w3
      { S7_Templates := "SrcType := Real" } NE_Contact(in1 := "Function Ratio check".PumpCaliberationControls."CurrentActual_A Gram", in2 := "actual_gramA_Old")
   END_RUNG wire#w4
   RUNG wire#w1
      Contact( "Function Ratio check".Control.AcceptValue )
      Move(in := 4, out1 => "RatioCheck_status")
   END_RUNG
   // the same network as SCL:
   #_w1 := "Functions"."2k"."mixing ratio program selected" AND "Function Ratio check".Control."Start metering" AND NOT "Temp".ratiocheck_temp[0];   // rising edge of "Function Ratio check".Control."Start metering"
   "Temp".ratiocheck_temp[0] := "Function Ratio check".Control."Start metering";
   IF #_w1 THEN "RatioCheck_status" := 1; END_IF;
   #_w2 := "Functions"."2k"."mixing ratio program selected" AND "Function Ratio check".Control."metering completed" AND NOT "Temp".ratiocheck_temp[1];   // rising edge of "Function Ratio check".Control."metering completed"
   "Temp".ratiocheck_temp[1] := "Function Ratio check".Control."metering completed";
   IF #_w2 THEN
       "RatioCheck_status" := 2;
       "actual_gramA_Old" := "Function Ratio check".PumpCaliberationControls."CurrentActual_A Gram";
       "actual_gramB_Old" := "Function Ratio check".PumpCaliberationControls."CurrentActual_B Gram";
   END_IF;
   #_w3 := "Functions"."2k"."mixing ratio program selected" AND ("Temp".ratiocheck_temp[3] OR "AlwaysTRUE") AND (("Function Ratio check".PumpCaliberationControls."CurrentActual_B Gram" <> "actual_gramB_Old") OR ("Function Ratio check".PumpCaliberationControls."CurrentActual_A Gram" <> "actual_gramA_Old"));
   #_w4 := #_w3 AND NOT "Temp".ratiocheck_temp[2];   // rising edge
   "Temp".ratiocheck_temp[2] := #_w3;
   IF #_w4 THEN "RatioCheck_status" := 3; END_IF;
   IF "Functions"."2k"."mixing ratio program selected" AND "Function Ratio check".Control.AcceptValue THEN
       "RatioCheck_status" := 4;
   END_IF;
END_REGION
END_FUNCTION

FUNCTION_BLOCK "FB3-Ratiocheck"   // FB3, LAD
{ S7_Optimized_Access := 'TRUE' }
VERSION : 0.1
// stored: AutoNumber false, IsIECCheckEnabled false, IsRetainMemResEnabled false, MemoryReserve 100, SetENOAutomatically false, UDAEnableTagReadback false
   VAR_INPUT
      Dispensing_time : DInt;
      "Set Qty in ml" : Real;
      "VC1 Pulses" : DInt;
      "VC2 Pulses" : DInt;
      VC1_impulse : Real;
      VC2_impulse : Real;
      "Outlet Open  to Pump ON A delay" : DInt;
      "Outlet Open  to Pump ON B delay" : DInt;
      "Pump Off  to Outlet Close" : DInt;
      "Pump Off  to Inlet A Close" : DInt;
      "Pump Off  to Inlet B Close" : DInt;
   END_VAR
   VAR_OUTPUT
      "Volume dispensed" : Real;
      "Run time" : Int;
   END_VAR
   VAR_IN_OUT
      ON_inlet_A : Bool;
      ON_inlet_B : Bool;
      ON_Pump_A : Bool;
      ON_pump_B : Bool;
      ON_valve_A : Bool;
      ON_valve_B : Bool;
      "Start Metering" : Bool;
      "Stop metering" : Bool;
      "Process running" : Bool;
      "process completed" : Bool;
   END_VAR
   VAR
      "pump A to valveA delay" : Bool;
      "Pump B to valve B delay" : Bool;
      "Pump Off to mixer off delay_1" : Bool;
      "VC1 pulses prev" : DInt;
      "VC2 pulses prev" : DInt;
      "VC1 pulse generted" : DInt;
      "VC2 pulse generated" : DInt;
      "Pump A Voulme dispensed" : Real;
      "Pump B volume dispensed" : Real;
      "Total Volume dispensed" : Real;
      "metering started" : Bool;
      "metering time in msec" : DInt;
      "dispense time elapsed" : Bool;
   END_VAR
   VAR_TEMP
      Ons_temp : Bool;
   END_VAR
   VAR_TEMP   // added for the SCL form of the ladder/FBD networks
      _w1 : Bool;
   END_VAR
BEGIN

REGION Network 1
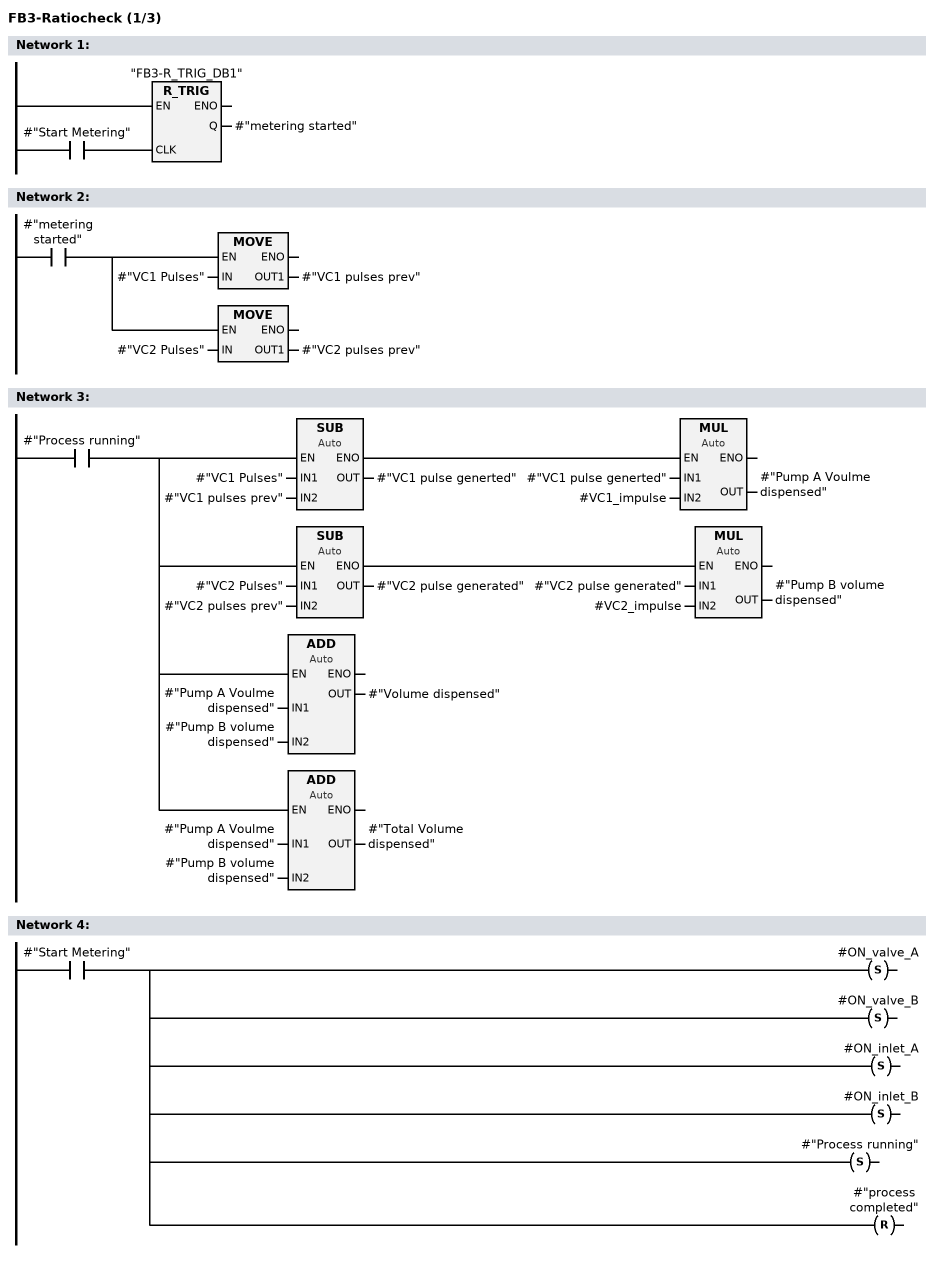
   RUNG wire#powerrail
      "FB3-R_TRIG_DB1".R_TRIG(CLK := wire#w1, Q => #"metering started")
   END_RUNG
   RUNG wire#powerrail
      Contact( #"Start Metering" )
   END_RUNG wire#w1
   // the same network as SCL:
   "FB3-R_TRIG_DB1"(CLK := #"Start Metering", Q => #"metering started");   // R_TRIG
END_REGION

REGION Network 2
   RUNG wire#powerrail
      Contact( #"metering started" )
      wire#w1
      Move(in := #"VC1 Pulses", out1 => #"VC1 pulses prev")
   END_RUNG
   RUNG wire#w1
      Move(in := #"VC2 Pulses", out1 => #"VC2 pulses prev")
   END_RUNG
   // the same network as SCL:
   IF #"metering started" THEN
       #"VC1 pulses prev" := #"VC1 Pulses";
       #"VC2 pulses prev" := #"VC2 Pulses";
   END_IF;
END_REGION

REGION Network 3
   RUNG wire#powerrail
      Contact( #"Process running" )
      wire#w1
      Sub(in1 := #"VC1 Pulses", in2 := #"VC1 pulses prev", out => #"VC1 pulse generted")
      Mul(in1 := #"VC1 pulse generted", in2 := #VC1_impulse, out => #"Pump A Voulme dispensed")
   END_RUNG
   RUNG wire#w1
      Sub(in1 := #"VC2 Pulses", in2 := #"VC2 pulses prev", out => #"VC2 pulse generated")
      Mul(in1 := #"VC2 pulse generated", in2 := #VC2_impulse, out => #"Pump B volume dispensed")
   END_RUNG
   RUNG wire#w1
      Add(in1 := #"Pump A Voulme dispensed", in2 := #"Pump B volume dispensed", out => #"Volume dispensed")
   END_RUNG
   RUNG wire#w1
      Add(in1 := #"Pump A Voulme dispensed", in2 := #"Pump B volume dispensed", out => #"Total Volume dispensed")
   END_RUNG
   // the same network as SCL:
   IF #"Process running" THEN
       #"VC1 pulse generted" := #"VC1 Pulses" - #"VC1 pulses prev";
       #"Pump A Voulme dispensed" := #"VC1 pulse generted" * #VC1_impulse;
       #"VC2 pulse generated" := #"VC2 Pulses" - #"VC2 pulses prev";
       #"Pump B volume dispensed" := #"VC2 pulse generated" * #VC2_impulse;
       #"Volume dispensed" := #"Pump A Voulme dispensed" + #"Pump B volume dispensed";
       #"Total Volume dispensed" := #"Pump A Voulme dispensed" + #"Pump B volume dispensed";
   END_IF;
END_REGION

REGION Network 4
   RUNG wire#powerrail
      Contact( #"Start Metering" )
      wire#w1
      S_Coil( #ON_valve_A )
   END_RUNG
   RUNG wire#w1
      S_Coil( #ON_valve_B )
   END_RUNG
   RUNG wire#w1
      S_Coil( #ON_inlet_A )
   END_RUNG
   RUNG wire#w1
      S_Coil( #ON_inlet_B )
   END_RUNG
   RUNG wire#w1
      S_Coil( #"Process running" )
   END_RUNG
   RUNG wire#w1
      R_Coil( #"process completed" )
   END_RUNG
   // the same network as SCL:
   IF #"Start Metering" THEN
       #ON_valve_A := TRUE;
       #ON_valve_B := TRUE;
       #ON_inlet_A := TRUE;
       #ON_inlet_B := TRUE;
       #"Process running" := TRUE;
       #"process completed" := FALSE;
   END_IF;
END_REGION

REGION Network 5
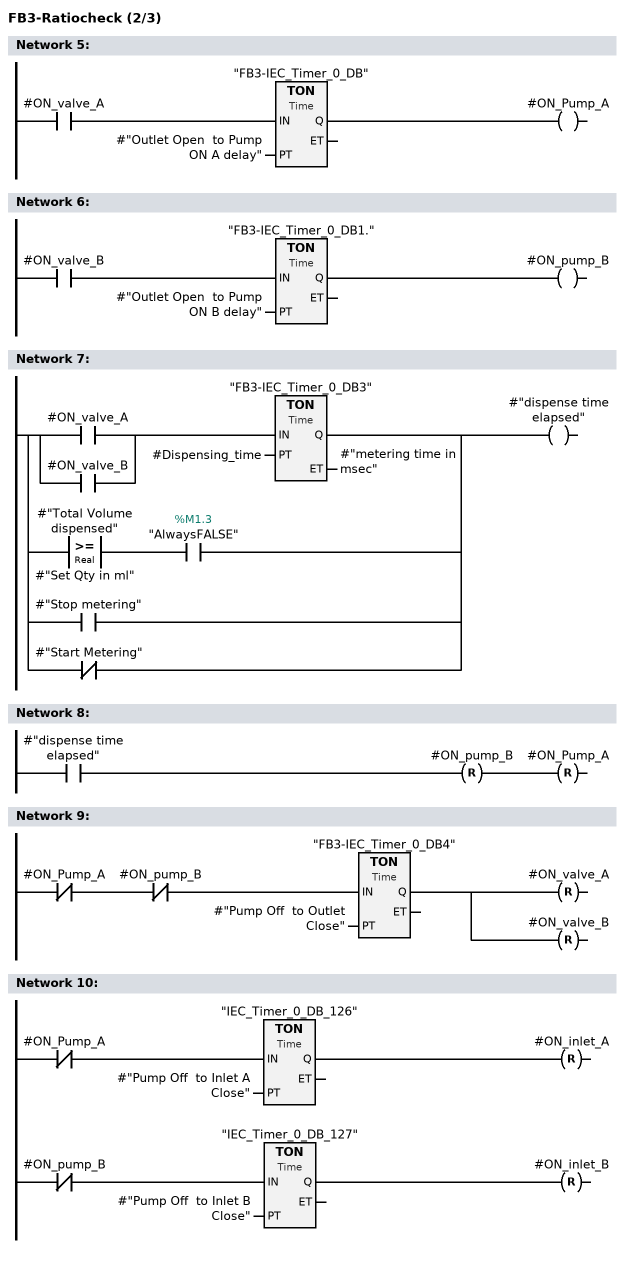
   RUNG wire#powerrail
      Contact( #ON_valve_A )
      { S7_Templates := "time_type := Time" } "FB3-IEC_Timer_0_DB".TON(pt := #"Outlet Open  to Pump ON A delay", et =>)
      Coil( #ON_Pump_A )
   END_RUNG
   // the same network as SCL:
   "FB3-IEC_Timer_0_DB".TON(IN := #ON_valve_A, PT := #"Outlet Open  to Pump ON A delay");
   #ON_Pump_A := "FB3-IEC_Timer_0_DB".Q;
END_REGION

REGION Network 6
   RUNG wire#powerrail
      Contact( #ON_valve_B )
      { S7_Templates := "time_type := Time" } "FB3-IEC_Timer_0_DB1.".TON(pt := #"Outlet Open  to Pump ON B delay", et =>)
      Coil( #ON_pump_B )
   END_RUNG
   // the same network as SCL:
   "FB3-IEC_Timer_0_DB1.".TON(IN := #ON_valve_B, PT := #"Outlet Open  to Pump ON B delay");
   #ON_pump_B := "FB3-IEC_Timer_0_DB1.".Q;
END_REGION

REGION Network 7
   RUNG wire#powerrail
      Contact( #ON_valve_A )
      wire#w1
      { S7_Templates := "time_type := Time" } "FB3-IEC_Timer_0_DB3".TON(pt := #Dispensing_time, et => #"metering time in msec")
      wire#w2
      Coil( #"dispense time elapsed" )
   END_RUNG
   RUNG wire#powerrail
      Contact( #ON_valve_B )
   END_RUNG wire#w1
   RUNG wire#powerrail
      { S7_Templates := "SrcType := Real" } GE_Contact(in1 := #"Total Volume dispensed", in2 := #"Set Qty in ml")
      Contact( "AlwaysFALSE" )
   END_RUNG wire#w2
   RUNG wire#powerrail
      Contact( #"Stop metering" )
   END_RUNG wire#w2
   RUNG wire#powerrail
      I_Contact( #"Start Metering" )
   END_RUNG wire#w2
   // the same network as SCL:
   "FB3-IEC_Timer_0_DB3".TON(IN := #ON_valve_A OR #ON_valve_B,
                           PT := #Dispensing_time,
                           ET => #"metering time in msec");
   #"dispense time elapsed" := "FB3-IEC_Timer_0_DB3".Q OR ((#"Total Volume dispensed" >= #"Set Qty in ml") AND "AlwaysFALSE") OR #"Stop metering" OR NOT #"Start Metering";
END_REGION

REGION Network 8
   RUNG wire#powerrail
      Contact( #"dispense time elapsed" )
      R_Coil( #ON_pump_B )
      R_Coil( #ON_Pump_A )
   END_RUNG
   // the same network as SCL:
   IF #"dispense time elapsed" THEN
       #ON_pump_B := FALSE;
       #ON_Pump_A := FALSE;
   END_IF;
END_REGION

REGION Network 9
   RUNG wire#powerrail
      I_Contact( #ON_Pump_A )
      I_Contact( #ON_pump_B )
      { S7_Templates := "time_type := Time" } "FB3-IEC_Timer_0_DB4".TON(pt := #"Pump Off  to Outlet Close", et =>)
      wire#w1
      R_Coil( #ON_valve_A )
   END_RUNG
   RUNG wire#w1
      R_Coil( #ON_valve_B )
   END_RUNG
   // the same network as SCL:
   "FB3-IEC_Timer_0_DB4".TON(IN := NOT #ON_Pump_A AND NOT #ON_pump_B, PT := #"Pump Off  to Outlet Close");
   IF "FB3-IEC_Timer_0_DB4".Q THEN
       #ON_valve_A := FALSE;
       #ON_valve_B := FALSE;
   END_IF;
END_REGION

REGION Network 10
   RUNG wire#powerrail
      I_Contact( #ON_Pump_A )
      { S7_Templates := "time_type := Time" } "IEC_Timer_0_DB_126".TON(pt := #"Pump Off  to Inlet A Close", et =>)
      R_Coil( #ON_inlet_A )
   END_RUNG
   RUNG wire#powerrail
      I_Contact( #ON_pump_B )
      { S7_Templates := "time_type := Time" } "IEC_Timer_0_DB_127".TON(pt := #"Pump Off  to Inlet B Close", et =>)
      R_Coil( #ON_inlet_B )
   END_RUNG
   // the same network as SCL:
   "IEC_Timer_0_DB_126".TON(IN := NOT #ON_Pump_A, PT := #"Pump Off  to Inlet A Close");
   IF "IEC_Timer_0_DB_126".Q THEN #ON_inlet_A := FALSE; END_IF;
   "IEC_Timer_0_DB_127".TON(IN := NOT #ON_pump_B, PT := #"Pump Off  to Inlet B Close");
   IF "IEC_Timer_0_DB_127".Q THEN #ON_inlet_B := FALSE; END_IF;
END_REGION

REGION Network 11
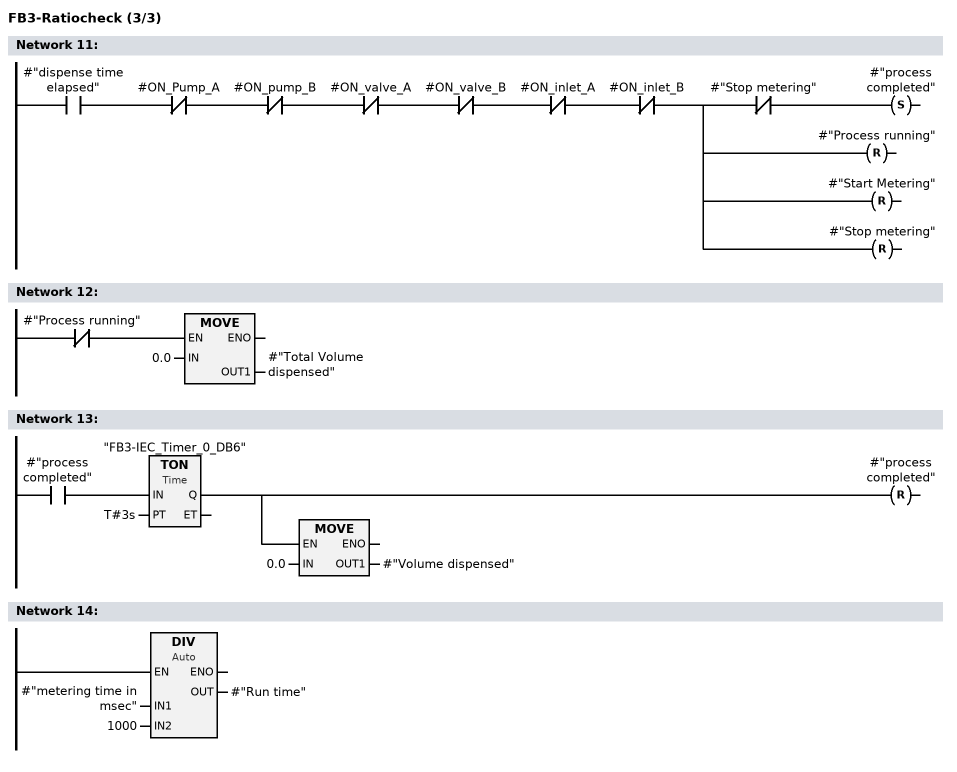
   RUNG wire#powerrail
      Contact( #"dispense time elapsed" )
      I_Contact( #ON_Pump_A )
      I_Contact( #ON_pump_B )
      I_Contact( #ON_valve_A )
      I_Contact( #ON_valve_B )
      I_Contact( #ON_inlet_A )
      I_Contact( #ON_inlet_B )
      wire#w1
      I_Contact( #"Stop metering" )
      S_Coil( #"process completed" )
   END_RUNG
   RUNG wire#w1
      R_Coil( #"Process running" )
   END_RUNG
   RUNG wire#w1
      R_Coil( #"Start Metering" )
   END_RUNG
   RUNG wire#w1
      R_Coil( #"Stop metering" )
   END_RUNG
   // the same network as SCL:
   #_w1 := #"dispense time elapsed" AND NOT #ON_Pump_A AND NOT #ON_pump_B AND NOT #ON_valve_A AND NOT #ON_valve_B AND NOT #ON_inlet_A AND NOT #ON_inlet_B;
   IF #_w1 AND NOT #"Stop metering" THEN #"process completed" := TRUE; END_IF;
   IF #_w1 THEN
       #"Process running" := FALSE;
       #"Start Metering" := FALSE;
       #"Stop metering" := FALSE;
   END_IF;
END_REGION

REGION Network 12
   RUNG wire#powerrail
      I_Contact( #"Process running" )
      Move(in := 0.0, out1 => #"Total Volume dispensed")
   END_RUNG
   // the same network as SCL:
   IF NOT #"Process running" THEN #"Total Volume dispensed" := 0.0; END_IF;
END_REGION

REGION Network 13
   RUNG wire#powerrail
      Contact( #"process completed" )
      { S7_Templates := "time_type := Time" } "FB3-IEC_Timer_0_DB6".TON(pt := T#3s, et =>)
      wire#w1
      R_Coil( #"process completed" )
   END_RUNG
   RUNG wire#w1
      Move(in := 0.0, out1 => #"Volume dispensed")
   END_RUNG
   // the same network as SCL:
   "FB3-IEC_Timer_0_DB6".TON(IN := #"process completed", PT := T#3s);
   IF "FB3-IEC_Timer_0_DB6".Q THEN
       #"process completed" := FALSE;
       #"Volume dispensed" := 0.0;
   END_IF;
END_REGION

REGION Network 14
   RUNG wire#powerrail
      Div(in1 := #"metering time in msec", in2 := 1000, out => #"Run time")
   END_RUNG
   // the same network as SCL:
   #"Run time" := #"metering time in msec" / 1000;
END_REGION
END_FUNCTION_BLOCK

FUNCTION "Faults" : Void   // FC25, LAD
{ S7_Optimized_Access := 'TRUE' }
VERSION : 0.1
// stored: AutoNumber true, IsIECCheckEnabled false, SetENOAutomatically false, UDAEnableTagReadback false
   VAR_TEMP
      spare3 : Bool;
   END_VAR
BEGIN

REGION Network 1
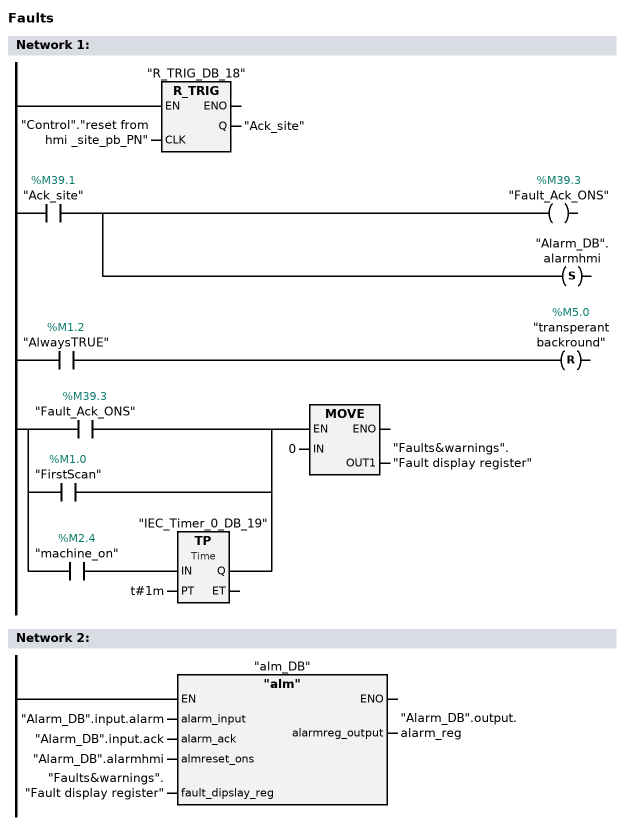
   RUNG wire#powerrail
      "R_TRIG_DB_18".R_TRIG(CLK := "Control"."reset from hmi _site_pb_PN", Q => "Ack_site")
   END_RUNG
   RUNG wire#powerrail
      Contact( "Ack_site" )
      wire#w1
      Coil( "Fault_Ack_ONS" )
   END_RUNG
   RUNG wire#w1
      S_Coil( "Alarm_DB".alarmhmi )
   END_RUNG
   RUNG wire#powerrail
      Contact( "AlwaysTRUE" )
      R_Coil( "transperant backround" )
   END_RUNG
   RUNG wire#powerrail
      Contact( "Fault_Ack_ONS" )
      wire#w2
      Move(in := 0, out1 => "Faults&warnings"."Fault display register")
   END_RUNG
   RUNG wire#powerrail
      Contact( "FirstScan" )
   END_RUNG wire#w2
   RUNG wire#powerrail
      Contact( "machine_on" )
      { S7_Templates := "time_type := Time" } "IEC_Timer_0_DB_19".TP(pt := t#1m, et =>)
   END_RUNG wire#w2
   // the same network as SCL:
   "R_TRIG_DB_18"(CLK := "Control"."reset from hmi _site_pb_PN", Q => "Ack_site");   // R_TRIG
   "Fault_Ack_ONS" := "Ack_site";
   IF "Ack_site" THEN "Alarm_DB".alarmhmi := TRUE; END_IF;
   IF "AlwaysTRUE" THEN "transperant backround" := FALSE; END_IF;
   "IEC_Timer_0_DB_19".TP(IN := "machine_on", PT := t#1m);
   IF "Fault_Ack_ONS" OR "FirstScan" OR "IEC_Timer_0_DB_19".Q THEN
       "Faults&warnings"."Fault display register" := 0;
   END_IF;
END_REGION

REGION Network 2
   RUNG wire#powerrail
      "alm_DB"(alarm_input := "Alarm_DB".input.alarm, alarm_ack := "Alarm_DB".input.ack, almreset_ons := "Alarm_DB".alarmhmi, fault_dipslay_reg := "Faults&warnings"."Fault display register", alarmreg_output => "Alarm_DB".output.alarm_reg)
   END_RUNG
   // the same network as SCL:
   "alm_DB"(alarm_input := "Alarm_DB".input.alarm,   // "alm"
            alarm_ack := "Alarm_DB".input.ack,
            almreset_ons := "Alarm_DB".alarmhmi,
            fault_dipslay_reg := "Faults&warnings"."Fault display register",
            alarmreg_output => "Alarm_DB".output.alarm_reg);
END_REGION

REGION Network 3 (SCL): Alarm FB call
   // "alm_DB"(alarm_input:=,
   //          alarmreg_output=>,
   //          alarm_ack:=,
   //          almreset_ons:=,
   //          fault_dipslay_reg:=);

   "Faults&warnings"."Fault present" := ("Faults&warnings"."Fault display register" <> 0); // fault present
   "Fault display register 1" := %DB36.;
   "Fault display register 2" := %DB36.;
   "Fault display register 3" := %DB36.;
   "Fault display register 4" := %DB36.;
   "Fault display register 5" := %DB36.;
   "Fault display register 6" := %DB36.;
END_REGION

REGION Network 4 (SCL): Alarm Register 1 ==== Fault Register 1
   "Alarm_DB".input.alarm[8] := NOT("emergency stop"); //A1-Emergenct stop active
   //"Alarm_DB".input.alarm[9] := "Faults&warnings"."Status Nok"."Drive controller A NK"; //A2-Pump A Drive Fault
   //"Alarm_DB".input.alarm[10] := "Faults&warnings"."Status Nok"."Drive controller B NK"; //A3-Pump B Drive Fault
   ////"Alarm_DB".input.alarm[11]:= agitatorA; //A4-Agitator A Fault
   ////"Alarm_DB".input.alarm[12]:= agitatorB; //A5-Agitator B Fault"
   // "Alarm_DB".input.alarm[13] := "Control".Level_sensor_enable AND ("Level Sensor A" >= 32767); //A6-Tank A level sensor fault
   // "Alarm_DB".input.alarm[14] := "Control".Level_sensor_enable AND ("Level Sensor B" >= 32767); //A7-Tank B level sensor fault
   // "Alarm_DB".input.alarm[15] := (("Control".Pressure_sensor_select = 0) AND ("Pressure sensor Pump Inlet A" >= 32767)) OR (("Control".Pressure_sensor_select = 1) AND ("Pressure sensor Pump Inlet A_mA" >= 32767));//A8-Pump A pressure sensor fault Inlet
   // "Alarm_DB".input.alarm[0] := (("Control".Pressure_sensor_select = 0) AND ("Pressure Sensor Pump Inlet B" >= 32767)) OR (("Control".Pressure_sensor_select = 1) AND ("Pressure Sensor Pump Inlet B_mA" >= 32767)); //A9-Pump B pressure sensor fault Inlet
   //"Alarm_DB".input.alarm[1] := "Re-filling Sequence DB"."Compare Re-fillingFilling sequence A"."Refilling Error";  //A10- Tank A refilling Error // not used
   //"Alarm_DB".input.alarm[2] := "Re-filling Sequence DB"."Compare Filling sequence b"."Refilling Error";  //A11- Tank B refilling Error // not used
   // "Alarm_DB".input.alarm[3] := NOT("heater status"."p100 connection okay".heater1) AND "Heater settings"."heater EN 1"; //A12-Heater1 sensor fault
   // "Alarm_DB".input.alarm[4] := NOT ("heater status"."p100 connection okay".heater2) AND "Heater settings"."heater EN 2";  //A13-Heater1 sensor fault
   // "Alarm_DB".input.alarm[5] := NOT ("heater status"."p100 connection okay".heater3) AND "Heater settings"."heater EN 3"; //A14-Heater3 sensor fault
   // "Alarm_DB".input.alarm[6] := NOT ("heater status"."p100 connection okay".heater4) AND "Heater settings"."heater EN 4";  //A15-Heater4 sensor fault
    //"Alarm_DB".input.alarm[7] := //A16-Reserve
END_REGION

REGION Network 5 (SCL): Alarm Register 2 ==== Fault Register 2
   // "Alarm_DB".input.alarm[24] := "heater status"."Limit under temperature".heater1; //"A17-Heater1 undertemperature" 
   // "Alarm_DB".input.alarm[25] := "heater status"."Limit under temperature".heater2; //A18-Heater2 undertemperature
   // "Alarm_DB".input.alarm[26] := "heater status"."Limit under temperature".heater3; //A19-Heater3 undertemperature
   // "Alarm_DB".input.alarm[27] := "heater status"."Limit under temperature".heater4; //A20-Heater4 undertemperature
   // "Alarm_DB".input.alarm[28] := "heater status"."Limit Over temperature".heater1; //"A21- Heater 1overtemperature"
   // "Alarm_DB".input.alarm[29] := "heater status"."Limit Over temperature".heater2; //"A22- Heater2 overtemperature"
   // "Alarm_DB".input.alarm[30] := "heater status"."Limit Over temperature".heater3; //"A23- Heater3 overtemperature"
   // "Alarm_DB".input.alarm[31] := "heater status"."Limit Over temperature".heater4; //"A24- Heater4 overtemperature"
    //"Alarm_DB".input.alarm[16] := //A25- Reserve
    //"Alarm_DB".input.alarm[17] := //A26- Reserve
    //"Alarm_DB".input.alarm[18] := //A27- Reserve
   // "Alarm_DB".input.alarm[19] := "Faults&warnings"."Status Nok"."Over pressure A inlet"; //A28- Pump A Inlet over pressure
   // "Alarm_DB".input.alarm[20] := "Faults&warnings"."Status Nok"."Over pressure B inlet"; //A29- Pump B Inlet over pressure
   // "Alarm_DB".input.alarm[21] := "Faults&warnings"."Status Nok"."Level empty A1" OR "Temp".bit20 ; //A30-Tank A1 Level Empty
   // //"Alarm_DB".input.alarm[22] := //A31-Reserve
   // "Alarm_DB".input.alarm[23] := "Faults&warnings"."Status Nok"."Level empty B1" OR "Temp".bit21; //A32-Tank B Level Empty
END_REGION

REGION Network 6 (SCL): Alarm Register 3 ==== Fault Register 3
   // "Alarm_DB".input.alarm[40] := "Faults&warnings"."Status Nok"."Low level A1"; //A33-Tank A1 low level 
   // //"Alarm_DB".input.alarm[41] :=  //A34-Reserve
   // "Alarm_DB".input.alarm[42] := "Faults&warnings"."Status Nok"."Low level B1"; //A35-Tank B low level
   // "Alarm_DB".input.alarm[43] := "pressure"."Control A"."under pressure Occured"; //A36-Pump A Inlet lower pressure
   // "Alarm_DB".input.alarm[44] := "pressure"."Control B"."under pressure Occured"; //A37-Pump B Inlet lower pressure
   // //"Alarm_DB".input.alarm[45] :=  //A38-Reserve
   // //"Alarm_DB".input.alarm[46] :=  //A39-Reserve
   "Alarm_DB".input.alarm[47] := "Potlife".contol."Potlife elapsed machine not in regeneration" AND NOT ("Functions"."2k"."pre run program selected") AND NOT ("Metering".Metering_running);  //A40-Potlife elapsed Change static mixer
    //"Alarm_DB".input.alarm[32] := //A41-Reserve
    //"Alarm_DB".input.alarm[33] := //A42-Reserve
    //"Alarm_DB".input.alarm[34] := //A43-Reserve
    //"Alarm_DB".input.alarm[35] := //A44-Reserve
    //"Alarm_DB".input.alarm[36] := //A45-Reserve
    //"Alarm_DB".input.alarm[37] := //A46-Reserve
   //"Alarm_DB".input.alarm[38] := //A47-Reserve
   //"Alarm_DB".input.alarm[39] := //A48-Reserve
END_REGION

REGION Network 7 (SCL): Alarm Register 4 ==== Fault Register 4
   //"Alarm_DB".input.alarm[56] :=  //A49-Reserve
   //"Alarm_DB".input.alarm[57] :=  //A50-Reserve
   //"Alarm_DB".input.alarm[58] := ///A51-Reserve
   //"Alarm_DB".input.alarm[59] := //A52-Reserve
   //"Alarm_DB".input.alarm[60] := //A53-Reserve
   //"Alarm_DB".input.alarm[61] :=  //A54-Reserve
   //"Alarm_DB".input.alarm[62] :=  //A55-Reserve
   //"Alarm_DB".input.alarm[63] := //A56-Reserve
    //"Alarm_DB".input.alarm[48] := //A57-Reserve
    //"Alarm_DB".input.alarm[49] := //A58-Reserve
    //"Alarm_DB".input.alarm[50] := //A59-Reserve
    //"Alarm_DB".input.alarm[51] := //A60-Reserve
    //"Alarm_DB".input.alarm[52] := //A61-Reserve
    //"Alarm_DB".input.alarm[53] := "Faults&warnings"."Status Nok"."Flowrate error"; //A62-Reserve
   //"Alarm_DB".input.alarm[54] := //A63-Reserve
   //"Alarm_DB".input.alarm[55] := //A64-Reserve
END_REGION

REGION Network 8 (SCL): Alarm Register 5 ==== Fault Register 5
   //"Alarm_DB".input.alarm[72] :=  //A65-Reserve
   //"Alarm_DB".input.alarm[73] :=  //A66-Reserve
   //"Alarm_DB".input.alarm[74] := ///A67-Reserve
   //"Alarm_DB".input.alarm[75] := //A68-Reserve
   //"Alarm_DB".input.alarm[76] := //A69-Reserve
   //"Alarm_DB".input.alarm[77] := "Mixing ratio"."mixing ratio Low Warning"; //A70-Warning mixing ratio low
   //"Alarm_DB".input.alarm[78] := "Mixing ratio"."mixing ratio high Warning"; //A71- warning Mixing Ratio high
   //"Alarm_DB".input.alarm[79] := "Mixing ratio"."Mixing ratio Low  Error"; //A72- Error Mixing ratio Low
   //"Alarm_DB".input.alarm[64] := "Mixing ratio"."Mixing ratio high Error"; //A73- Error Mixing Ratio high
    //"Alarm_DB".input.alarm[65] := //A74-Reserve
    //"Alarm_DB".input.alarm[66] := //A75-Reserve
    //"Alarm_DB".input.alarm[67] := //A76-Reserve
    //"Alarm_DB".input.alarm[68] := //A77-Reserve
    //"Alarm_DB".input.alarm[69] := //A78-Reserve
   //"Alarm_DB".input.alarm[70] := //A79-Reserve
   //"Alarm_DB".input.alarm[71] := //A80-Reserve
END_REGION

REGION Network 9 (SCL): Alarm Register 6 ==== Fault Register 6
   // //"Alarm_DB".input.alarm[88] := //A81-Reserve
   // "Alarm_DB".input.alarm[89] := "level"."Drum Level Low A1"; //"A82-Level Low Drum A1"
   // "Alarm_DB".input.alarm[90] := "level"."Drum Level Low B1"; //"A83-Level Low Drum B1"
   // "Alarm_DB".input.alarm[91] := "level"."Drum Level Low A2"; //"A84-Level Low Drum A2"
   // "Alarm_DB".input.alarm[92] := "level"."Drum Level Low B2"; //"A85-Level Low Drum B2"
   // "Alarm_DB".input.alarm[93] := "level"."Drum Level Empty A1"; //"A86-Level Empty Drum A1"
   // "Alarm_DB".input.alarm[94] := "level"."Drum Level Empty B1";//"A87-Level Empty Drum B1"
   // "Alarm_DB".input.alarm[95] := "level"."Drum Level Empty A2"; //"A88-Level Empty Drum A2"
   // "Alarm_DB".input.alarm[80] := "level"."Drum Level Empty B2"; //"A89-Level Empty Drum B2"
   // "Temp".bit20 := ("HMI".supplySelection = 1) AND "level"."Drum Level Empty A1" AND "level"."Drum Level Empty A2";
   // "Temp".bit21 := ("HMI".supplySelection = 1) AND "level"."Drum Level Empty B1" AND "level"."Drum Level Empty B2";
   // "Alarm_DB".input.alarm[81] := "Faults&warnings"."Status Nok"."Pressure sensor Pump A Outlet"; //"A90 Pressure sensor Pump A Outlet Fault"
   // "Alarm_DB".input.alarm[82] := "Faults&warnings"."Status Nok"."Pressure Sensor Pump B Outlet"; //"A91 Pressure sensor Pump B Outlet Fault"
   // "Alarm_DB".input.alarm[83] := "Faults&warnings"."Status Nok"."Over pressure A outlet"; //A92- Pump A Outlet Over PRessure
   // "Alarm_DB".input.alarm[84] := "Faults&warnings"."Status Nok"."Over pressure B outlet"; //"A93 Over pressure B outlet"
   // "Alarm_DB".input.alarm[85] := "pressure"."Control A_Outlet"."under pressure Occured"; //A94- Pump A Outlet Under Pressure
   // "Alarm_DB".input.alarm[86] := "pressure"."Control B_Outlet"."under pressure Occured"; //"A95- Pump B Outlet Under Pressure"
   // //"Alarm_DB".input.alarm[87] := //A96-Reserve
END_REGION
END_FUNCTION

FUNCTION_BLOCK "alm"   // FB4, LAD
{ S7_Optimized_Access := 'TRUE' }
VERSION : 0.1
// stored: AutoNumber true, IsIECCheckEnabled false, IsRetainMemResEnabled false, MemoryReserve 100, SetENOAutomatically false, UDAEnableTagReadback false
   VAR_INPUT
      alarm_input : Array[0..95] of Bool;
   END_VAR
   VAR_OUTPUT
      alarmreg_output : Array[0..95] of Bool;
   END_VAR
   VAR_IN_OUT
      alarm_ack : Array[0..95] of Bool;
      almreset_ons : Bool;
      fault_dipslay_reg : Int;
   END_VAR
   VAR
      i : Int;
      alarmregtemp : Array[0..95] of Bool;
      temp : Array[0..95] of Bool;
   END_VAR
   VAR_TEMP   // added for the SCL form of the ladder/FBD networks
      _w1 : Bool;
      _w2 : Bool;
      _w3 : Bool;
   END_VAR
BEGIN

REGION Network 1
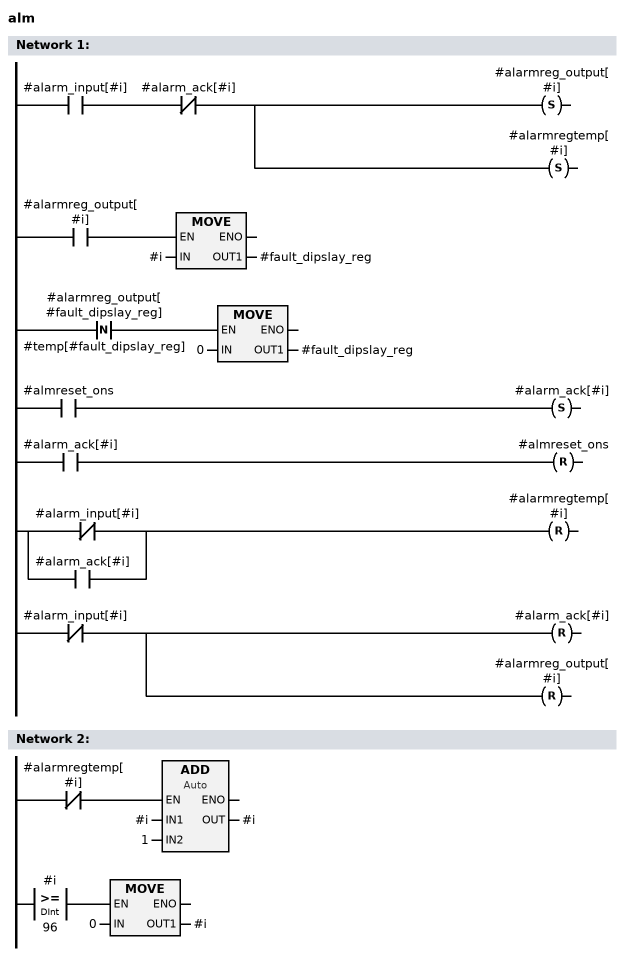
   RUNG wire#powerrail
      Contact( #alarm_input[#i] )
      I_Contact( #alarm_ack[#i] )
      wire#w1
      S_Coil( #alarmreg_output[#i] )
   END_RUNG
   RUNG wire#w1
      S_Coil( #alarmregtemp[#i] )
   END_RUNG
   RUNG wire#powerrail
      Contact( #alarmreg_output[#i] )
      Move(in := #i, out1 => #fault_dipslay_reg)
   END_RUNG
   RUNG wire#powerrail
      N_Contact(operand := #alarmreg_output[#fault_dipslay_reg], bit := #temp[#fault_dipslay_reg])
      Move(in := 0, out1 => #fault_dipslay_reg)
   END_RUNG
   RUNG wire#powerrail
      Contact( #almreset_ons )
      S_Coil( #alarm_ack[#i] )
   END_RUNG
   RUNG wire#powerrail
      Contact( #alarm_ack[#i] )
      R_Coil( #almreset_ons )
   END_RUNG
   RUNG wire#powerrail
      I_Contact( #alarm_input[#i] )
      wire#w2
      R_Coil( #alarmregtemp[#i] )
   END_RUNG
   RUNG wire#powerrail
      Contact( #alarm_ack[#i] )
   END_RUNG wire#w2
   RUNG wire#powerrail
      I_Contact( #alarm_input[#i] )
      wire#w3
      R_Coil( #alarm_ack[#i] )
   END_RUNG
   RUNG wire#w3
      R_Coil( #alarmreg_output[#i] )
   END_RUNG
   // the same network as SCL:
   #_w1 := #alarm_input[#i] AND NOT #alarm_ack[#i];
   IF #_w1 THEN
       #alarmreg_output[#i] := TRUE;
       #alarmregtemp[#i] := TRUE;
   END_IF;
   IF #alarmreg_output[#i] THEN #fault_dipslay_reg := #i; END_IF;
   #_w2 := NOT #alarmreg_output[#fault_dipslay_reg] AND #temp[#fault_dipslay_reg];   // falling edge of #alarmreg_output[#fault_dipslay_reg]
   #temp[#fault_dipslay_reg] := #alarmreg_output[#fault_dipslay_reg];
   IF #_w2 THEN #fault_dipslay_reg := 0; END_IF;
   IF #almreset_ons THEN #alarm_ack[#i] := TRUE; END_IF;
   IF #alarm_ack[#i] THEN #almreset_ons := FALSE; END_IF;
   IF NOT #alarm_input[#i] OR #alarm_ack[#i] THEN #alarmregtemp[#i] := FALSE; END_IF;
   #_w3 := NOT #alarm_input[#i];
   IF #_w3 THEN
       #alarm_ack[#i] := FALSE;
       #alarmreg_output[#i] := FALSE;
   END_IF;
END_REGION

REGION Network 2
   RUNG wire#powerrail
      I_Contact( #alarmregtemp[#i] )
      Add(in1 := #i, in2 := 1, out => #i)
   END_RUNG
   RUNG wire#powerrail
      { S7_Templates := "SrcType := DInt" } GE_Contact(in1 := #i, in2 := 96)
      Move(in := 0, out1 => #i)
   END_RUNG
   // the same network as SCL:
   IF NOT #alarmregtemp[#i] THEN #i := #i + 1; END_IF;
   IF #i >= 96 THEN #i := 0; END_IF;
END_REGION
END_FUNCTION_BLOCK

FUNCTION "Flowrate FC" : Void   // FC35, LAD
{ S7_Optimized_Access := 'TRUE' }
VERSION : 0.1
// stored: AutoNumber true, IsIECCheckEnabled false, SetENOAutomatically false, UDAEnableTagReadback false
BEGIN

REGION Network 1: Pump size according to ml/l/kg
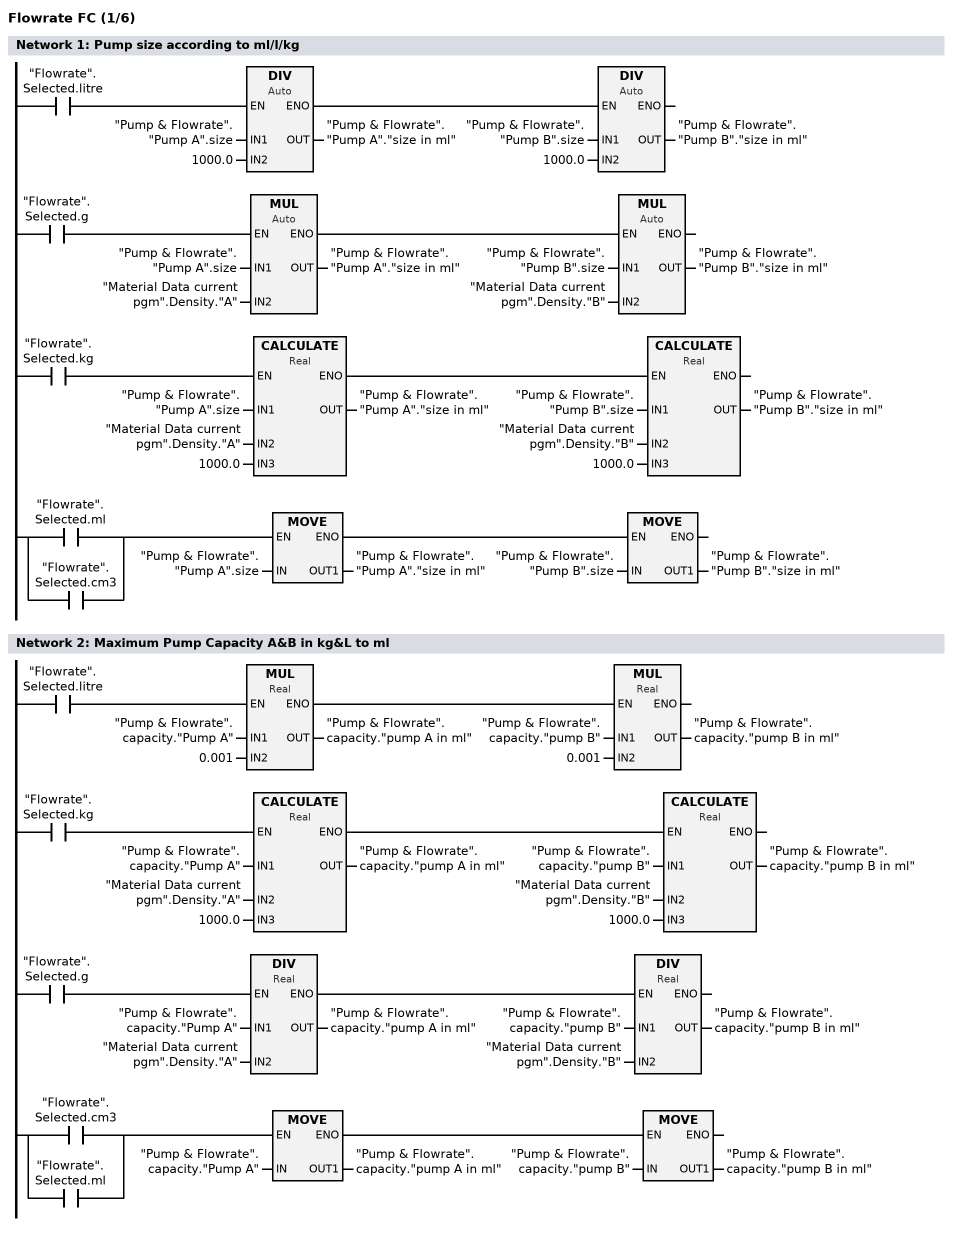
   IF "Flowrate".Selected.litre THEN
       "Pump & Flowrate"."Pump A"."size in ml" := "Pump & Flowrate"."Pump A".size / 1000.0;
       "Pump & Flowrate"."Pump B"."size in ml" := "Pump & Flowrate"."Pump B".size / 1000.0;
   END_IF;
   IF "Flowrate".Selected.g THEN
       "Pump & Flowrate"."Pump A"."size in ml" := "Pump & Flowrate"."Pump A".size * "Material Data current pgm".Density."A";
       "Pump & Flowrate"."Pump B"."size in ml" := "Pump & Flowrate"."Pump B".size * "Material Data current pgm".Density."B";
   END_IF;
   IF "Flowrate".Selected.kg THEN
       "Pump & Flowrate"."Pump A"."size in ml" := ("Pump & Flowrate"."Pump A".size*"Material Data current pgm".Density."A")/1000.0;
       "Pump & Flowrate"."Pump B"."size in ml" := ("Pump & Flowrate"."Pump B".size*"Material Data current pgm".Density."B")/1000.0;
   END_IF;
   IF "Flowrate".Selected.ml OR "Flowrate".Selected.cm3 THEN
       "Pump & Flowrate"."Pump A"."size in ml" := "Pump & Flowrate"."Pump A".size;
       "Pump & Flowrate"."Pump B"."size in ml" := "Pump & Flowrate"."Pump B".size;
   END_IF;
END_REGION

REGION Network 2: Maximum Pump Capacity A&B in kg&L to ml
   IF "Flowrate".Selected.litre THEN
       "Pump & Flowrate".capacity."pump A in ml" := "Pump & Flowrate".capacity."Pump A" * 0.001;
       "Pump & Flowrate".capacity."pump B in ml" := "Pump & Flowrate".capacity."pump B" * 0.001;
   END_IF;
   IF "Flowrate".Selected.kg THEN
       "Pump & Flowrate".capacity."pump A in ml" := ("Pump & Flowrate".capacity."Pump A"*"Material Data current pgm".Density."A")/1000.0;
       "Pump & Flowrate".capacity."pump B in ml" := ("Pump & Flowrate".capacity."pump B"*"Material Data current pgm".Density."B")/1000.0;
   END_IF;
   IF "Flowrate".Selected.g THEN
       "Pump & Flowrate".capacity."pump A in ml" := "Pump & Flowrate".capacity."Pump A" / "Material Data current pgm".Density."A";
       "Pump & Flowrate".capacity."pump B in ml" := "Pump & Flowrate".capacity."pump B" / "Material Data current pgm".Density."B";
   END_IF;
   IF "Flowrate".Selected.cm3 OR "Flowrate".Selected.ml THEN
       "Pump & Flowrate".capacity."pump A in ml" := "Pump & Flowrate".capacity."Pump A";
       "Pump & Flowrate".capacity."pump B in ml" := "Pump & Flowrate".capacity."pump B";
   END_IF;
END_REGION

REGION Network 3: Mixed flowrate Minimum
   // 10% of maximum Flowrate
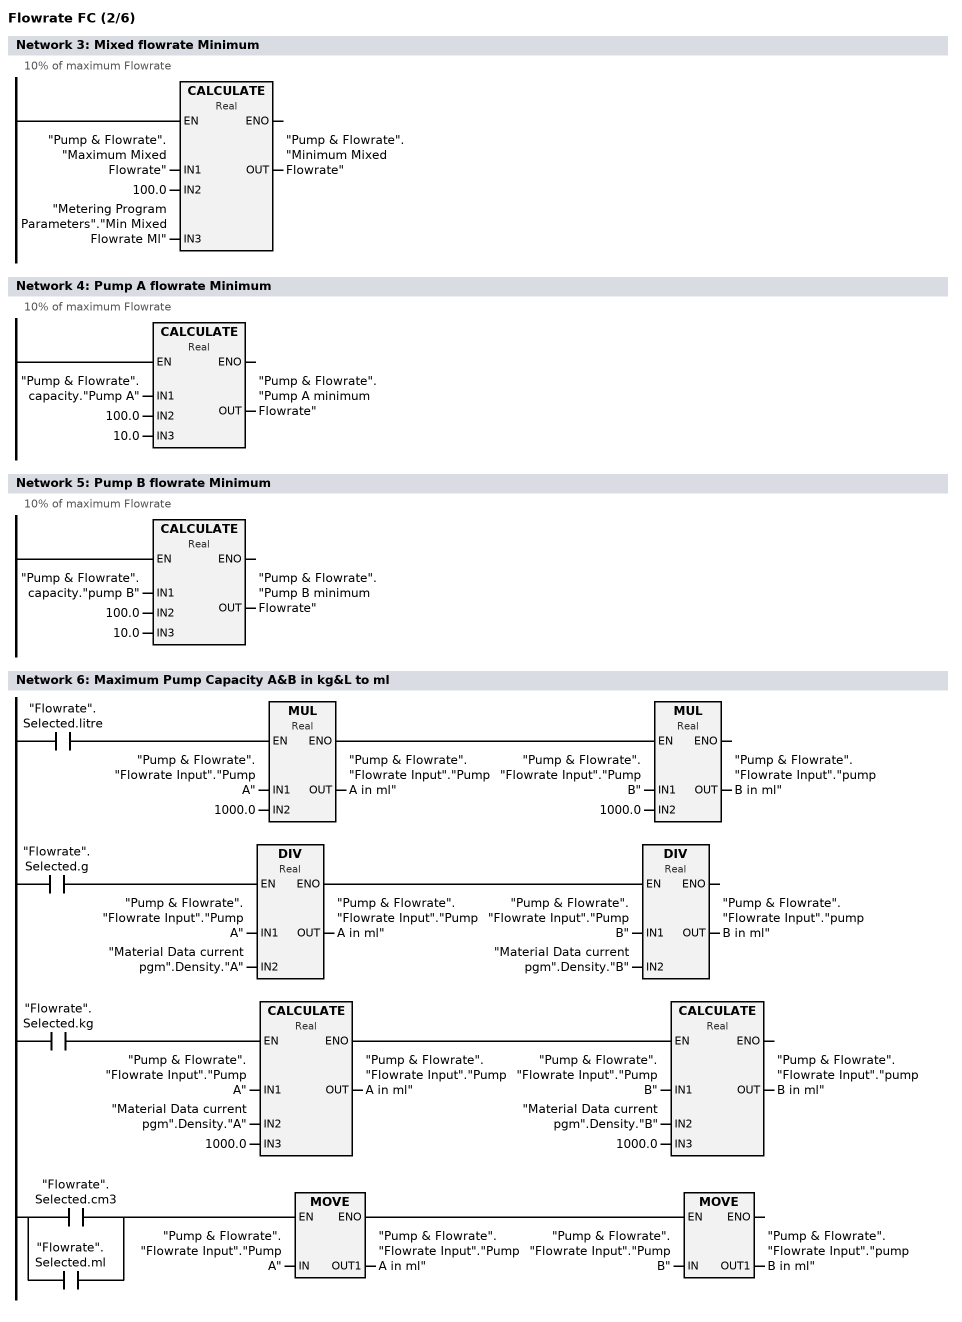
   "Pump & Flowrate"."Minimum Mixed Flowrate" := ("Pump & Flowrate"."Maximum Mixed Flowrate"/100.0)*"Metering Program Parameters"."Min Mixed Flowrate Ml";
END_REGION

REGION Network 4: Pump A flowrate Minimum
   // 10% of maximum Flowrate
   "Pump & Flowrate"."Pump A minimum Flowrate" := ("Pump & Flowrate".capacity."Pump A"/100.0)*10.0;
END_REGION

REGION Network 5: Pump B flowrate Minimum
   // 10% of maximum Flowrate
   "Pump & Flowrate"."Pump B minimum Flowrate" := ("Pump & Flowrate".capacity."pump B"/100.0)*10.0;
END_REGION

REGION Network 6: Maximum Pump Capacity A&B in kg&L to ml
   IF "Flowrate".Selected.litre THEN
       "Pump & Flowrate"."Flowrate Input"."Pump A in ml" := "Pump & Flowrate"."Flowrate Input"."Pump A" * 1000.0;
       "Pump & Flowrate"."Flowrate Input"."pump B in ml" := "Pump & Flowrate"."Flowrate Input"."Pump B" * 1000.0;
   END_IF;
   IF "Flowrate".Selected.g THEN
       "Pump & Flowrate"."Flowrate Input"."Pump A in ml" := "Pump & Flowrate"."Flowrate Input"."Pump A" / "Material Data current pgm".Density."A";
       "Pump & Flowrate"."Flowrate Input"."pump B in ml" := "Pump & Flowrate"."Flowrate Input"."Pump B" / "Material Data current pgm".Density."B";
   END_IF;
   IF "Flowrate".Selected.kg THEN
       "Pump & Flowrate"."Flowrate Input"."Pump A in ml" := ("Pump & Flowrate"."Flowrate Input"."Pump A"*"Material Data current pgm".Density."A")/1000.0;
       "Pump & Flowrate"."Flowrate Input"."pump B in ml" := ("Pump & Flowrate"."Flowrate Input"."Pump B"*"Material Data current pgm".Density."B")/1000.0;
   END_IF;
   IF "Flowrate".Selected.cm3 OR "Flowrate".Selected.ml THEN
       "Pump & Flowrate"."Flowrate Input"."Pump A in ml" := "Pump & Flowrate"."Flowrate Input"."Pump A";
       "Pump & Flowrate"."Flowrate Input"."pump B in ml" := "Pump & Flowrate"."Flowrate Input"."Pump B";
   END_IF;
END_REGION

REGION Network 7: Current Flowrate A In ml/litre/kg
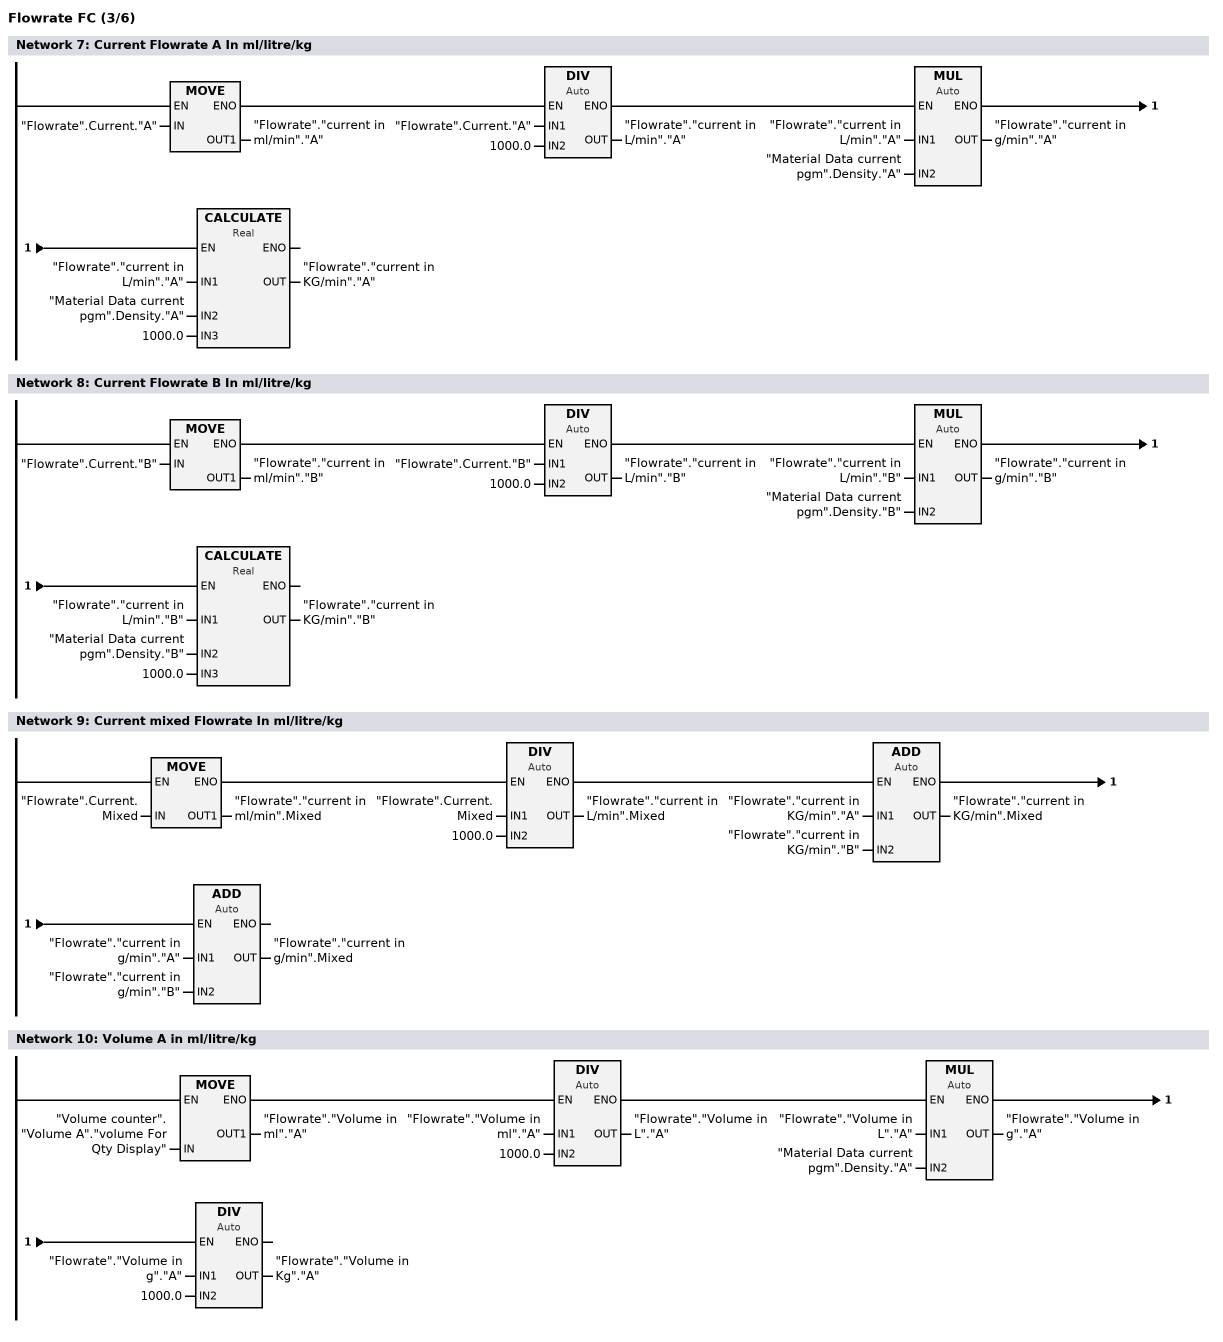
   RUNG wire#powerrail
      Move(in := "Flowrate".Current."A", out1 => "Flowrate"."current in ml/min"."A")
      Div(in1 := "Flowrate".Current."A", in2 := 1000.0, out => "Flowrate"."current in L/min"."A")
      Mul(in1 := "Flowrate"."current in L/min"."A", in2 := "Material Data current pgm".Density."A", out => "Flowrate"."current in g/min"."A")
      { S7_Templates := "SrcType := Real"; S7_Expression := "(IN1*IN2)/IN3" } Calculate(in1 := "Flowrate"."current in L/min"."A", in2 := "Material Data current pgm".Density."A", in3 := 1000.0, out => "Flowrate"."current in KG/min"."A")
   END_RUNG
   // the same network as SCL:
   "Flowrate"."current in ml/min"."A" := "Flowrate".Current."A";
   "Flowrate"."current in L/min"."A" := "Flowrate".Current."A" / 1000.0;
   "Flowrate"."current in g/min"."A" := "Flowrate"."current in L/min"."A" * "Material Data current pgm".Density."A";
   "Flowrate"."current in KG/min"."A" := ("Flowrate"."current in L/min"."A"*"Material Data current pgm".Density."A")/1000.0;
END_REGION

REGION Network 8: Current Flowrate B In ml/litre/kg
   RUNG wire#powerrail
      Move(in := "Flowrate".Current."B", out1 => "Flowrate"."current in ml/min"."B")
      Div(in1 := "Flowrate".Current."B", in2 := 1000.0, out => "Flowrate"."current in L/min"."B")
      Mul(in1 := "Flowrate"."current in L/min"."B", in2 := "Material Data current pgm".Density."B", out => "Flowrate"."current in g/min"."B")
      { S7_Templates := "SrcType := Real"; S7_Expression := "(IN1*IN2)/IN3" } Calculate(in1 := "Flowrate"."current in L/min"."B", in2 := "Material Data current pgm".Density."B", in3 := 1000.0, out => "Flowrate"."current in KG/min"."B")
   END_RUNG
   // the same network as SCL:
   "Flowrate"."current in ml/min"."B" := "Flowrate".Current."B";
   "Flowrate"."current in L/min"."B" := "Flowrate".Current."B" / 1000.0;
   "Flowrate"."current in g/min"."B" := "Flowrate"."current in L/min"."B" * "Material Data current pgm".Density."B";
   "Flowrate"."current in KG/min"."B" := ("Flowrate"."current in L/min"."B"*"Material Data current pgm".Density."B")/1000.0;
END_REGION

REGION Network 9: Current mixed Flowrate In ml/litre/kg
   RUNG wire#powerrail
      Move(in := "Flowrate".Current.Mixed, out1 => "Flowrate"."current in ml/min".Mixed)
      Div(in1 := "Flowrate".Current.Mixed, in2 := 1000.0, out => "Flowrate"."current in L/min".Mixed)
      Add(in1 := "Flowrate"."current in KG/min"."A", in2 := "Flowrate"."current in KG/min"."B", out => "Flowrate"."current in KG/min".Mixed)
      Add(in1 := "Flowrate"."current in g/min"."A", in2 := "Flowrate"."current in g/min"."B", out => "Flowrate"."current in g/min".Mixed)
   END_RUNG
   // the same network as SCL:
   "Flowrate"."current in ml/min".Mixed := "Flowrate".Current.Mixed;
   "Flowrate"."current in L/min".Mixed := "Flowrate".Current.Mixed / 1000.0;
   "Flowrate"."current in KG/min".Mixed := "Flowrate"."current in KG/min"."A" + "Flowrate"."current in KG/min"."B";
   "Flowrate"."current in g/min".Mixed := "Flowrate"."current in g/min"."A" + "Flowrate"."current in g/min"."B";
END_REGION

REGION Network 10: Volume A in ml/litre/kg
   RUNG wire#powerrail
      Move(in := "Volume counter"."Volume A"."volume For Qty Display", out1 => "Flowrate"."Volume in ml"."A")
      Div(in1 := "Flowrate"."Volume in ml"."A", in2 := 1000.0, out => "Flowrate"."Volume in L"."A")
      Mul(in1 := "Flowrate"."Volume in L"."A", in2 := "Material Data current pgm".Density."A", out => "Flowrate"."Volume in g"."A")
      Div(in1 := "Flowrate"."Volume in g"."A", in2 := 1000.0, out => "Flowrate"."Volume in Kg"."A")
   END_RUNG
   // the same network as SCL:
   "Flowrate"."Volume in ml"."A" := "Volume counter"."Volume A"."volume For Qty Display";
   "Flowrate"."Volume in L"."A" := "Flowrate"."Volume in ml"."A" / 1000.0;
   "Flowrate"."Volume in g"."A" := "Flowrate"."Volume in L"."A" * "Material Data current pgm".Density."A";
   "Flowrate"."Volume in Kg"."A" := "Flowrate"."Volume in g"."A" / 1000.0;
END_REGION

REGION Network 11: Volume B in ml/litre/kg
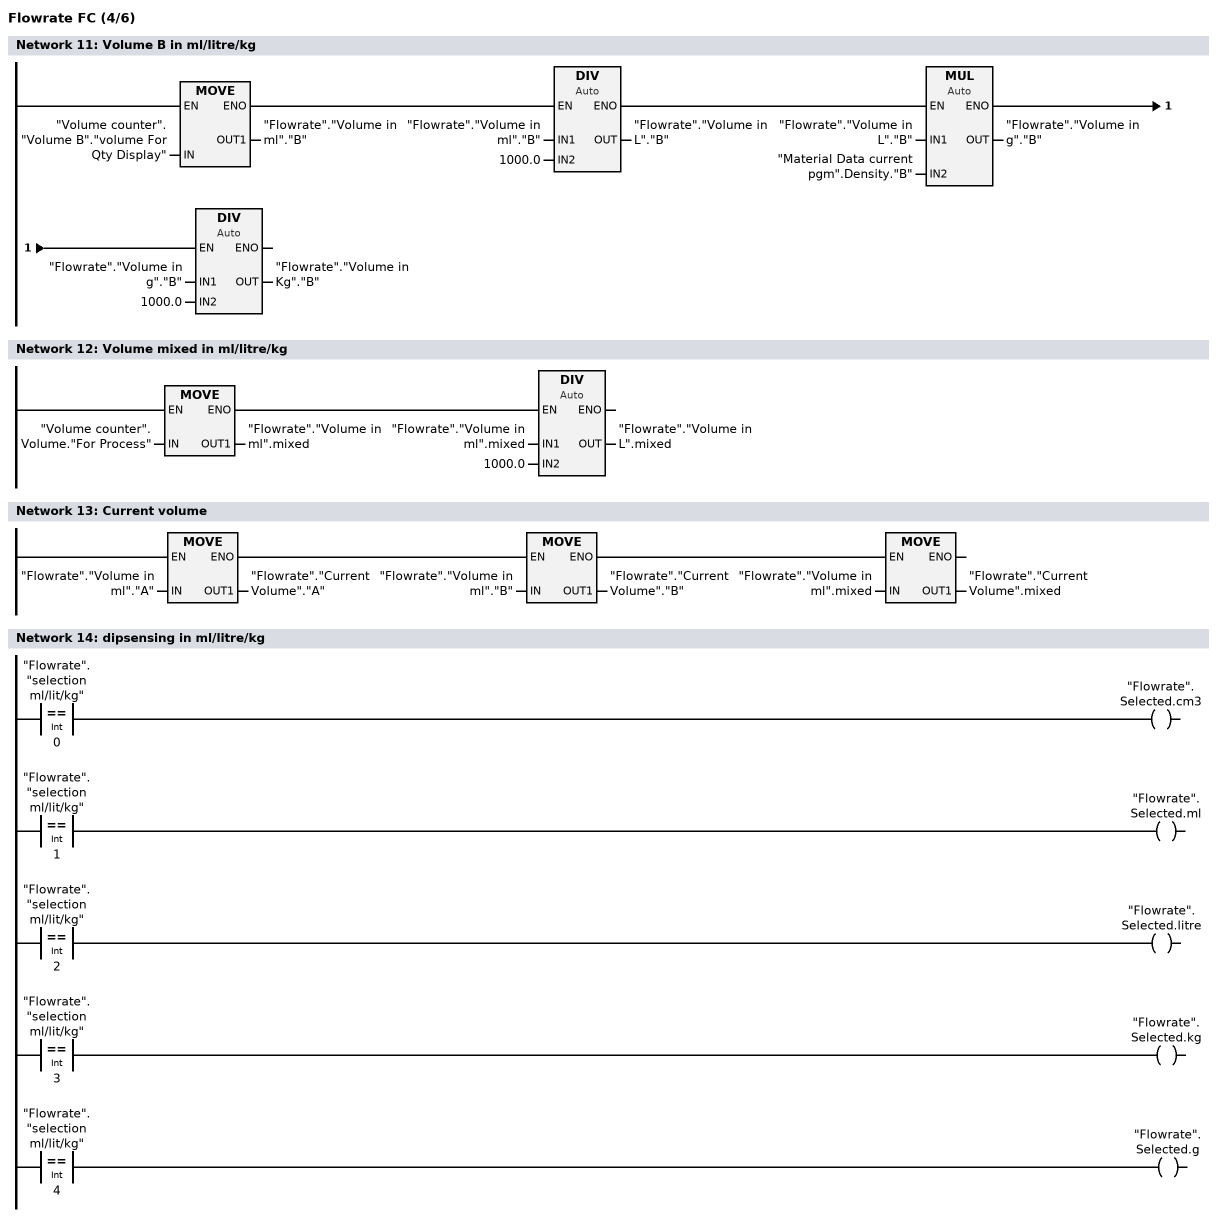
   RUNG wire#powerrail
      Move(in := "Volume counter"."Volume B"."volume For Qty Display", out1 => "Flowrate"."Volume in ml"."B")
      Div(in1 := "Flowrate"."Volume in ml"."B", in2 := 1000.0, out => "Flowrate"."Volume in L"."B")
      Mul(in1 := "Flowrate"."Volume in L"."B", in2 := "Material Data current pgm".Density."B", out => "Flowrate"."Volume in g"."B")
      Div(in1 := "Flowrate"."Volume in g"."B", in2 := 1000.0, out => "Flowrate"."Volume in Kg"."B")
   END_RUNG
   // the same network as SCL:
   "Flowrate"."Volume in ml"."B" := "Volume counter"."Volume B"."volume For Qty Display";
   "Flowrate"."Volume in L"."B" := "Flowrate"."Volume in ml"."B" / 1000.0;
   "Flowrate"."Volume in g"."B" := "Flowrate"."Volume in L"."B" * "Material Data current pgm".Density."B";
   "Flowrate"."Volume in Kg"."B" := "Flowrate"."Volume in g"."B" / 1000.0;
END_REGION

REGION Network 12: Volume mixed in ml/litre/kg
   RUNG wire#powerrail
      Move(in := "Volume counter".Volume."For Process", out1 => "Flowrate"."Volume in ml".mixed)
      Div(in1 := "Flowrate"."Volume in ml".mixed, in2 := 1000.0, out => "Flowrate"."Volume in L".mixed)
   END_RUNG
   // the same network as SCL:
   "Flowrate"."Volume in ml".mixed := "Volume counter".Volume."For Process";
   "Flowrate"."Volume in L".mixed := "Flowrate"."Volume in ml".mixed / 1000.0;
END_REGION

REGION Network 13: Current volume
   RUNG wire#powerrail
      Move(in := "Flowrate"."Volume in ml"."A", out1 => "Flowrate"."Current Volume"."A")
      Move(in := "Flowrate"."Volume in ml"."B", out1 => "Flowrate"."Current Volume"."B")
      Move(in := "Flowrate"."Volume in ml".mixed, out1 => "Flowrate"."Current Volume".mixed)
   END_RUNG
   // the same network as SCL:
   "Flowrate"."Current Volume"."A" := "Flowrate"."Volume in ml"."A";
   "Flowrate"."Current Volume"."B" := "Flowrate"."Volume in ml"."B";
   "Flowrate"."Current Volume".mixed := "Flowrate"."Volume in ml".mixed;
END_REGION

REGION Network 14: dipsensing in ml/litre/kg
   RUNG wire#powerrail
      { S7_Templates := "SrcType := Int" } EQ_Contact(in1 := "Flowrate"."selection ml/lit/kg", in2 := 0)
      Coil( "Flowrate".Selected.cm3 )
   END_RUNG
   RUNG wire#powerrail
      { S7_Templates := "SrcType := Int" } EQ_Contact(in1 := "Flowrate"."selection ml/lit/kg", in2 := 1)
      Coil( "Flowrate".Selected.ml )
   END_RUNG
   RUNG wire#powerrail
      { S7_Templates := "SrcType := Int" } EQ_Contact(in1 := "Flowrate"."selection ml/lit/kg", in2 := 2)
      Coil( "Flowrate".Selected.litre )
   END_RUNG
   RUNG wire#powerrail
      { S7_Templates := "SrcType := Int" } EQ_Contact(in1 := "Flowrate"."selection ml/lit/kg", in2 := 3)
      Coil( "Flowrate".Selected.kg )
   END_RUNG
   RUNG wire#powerrail
      { S7_Templates := "SrcType := Int" } EQ_Contact(in1 := "Flowrate"."selection ml/lit/kg", in2 := 4)
      Coil( "Flowrate".Selected.g )
   END_RUNG
   // the same network as SCL:
   "Flowrate".Selected.cm3 := "Flowrate"."selection ml/lit/kg" = 0;
   "Flowrate".Selected.ml := "Flowrate"."selection ml/lit/kg" = 1;
   "Flowrate".Selected.litre := "Flowrate"."selection ml/lit/kg" = 2;
   "Flowrate".Selected.kg := "Flowrate"."selection ml/lit/kg" = 3;
   "Flowrate".Selected.g := "Flowrate"."selection ml/lit/kg" = 4;
END_REGION

REGION Network 15: Display flowrate in ml
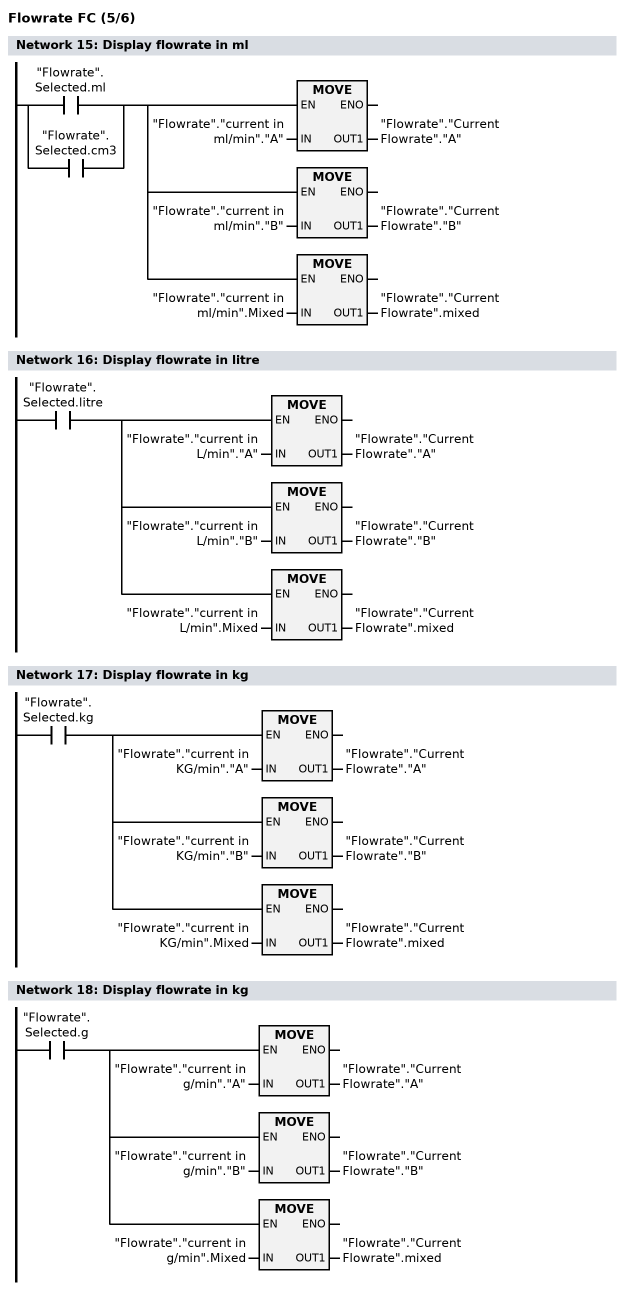
   RUNG wire#powerrail
      Contact( "Flowrate".Selected.ml )
      wire#w1
      Move(in := "Flowrate"."current in ml/min"."A", out1 => "Flowrate"."Current Flowrate"."A")
   END_RUNG
   RUNG wire#powerrail
      Contact( "Flowrate".Selected.cm3 )
   END_RUNG wire#w1
   RUNG wire#w1
      Move(in := "Flowrate"."current in ml/min"."B", out1 => "Flowrate"."Current Flowrate"."B")
   END_RUNG
   RUNG wire#w1
      Move(in := "Flowrate"."current in ml/min".Mixed, out1 => "Flowrate"."Current Flowrate".mixed)
   END_RUNG
   // the same network as SCL:
   IF "Flowrate".Selected.ml OR "Flowrate".Selected.cm3 THEN
       "Flowrate"."Current Flowrate"."A" := "Flowrate"."current in ml/min"."A";
       "Flowrate"."Current Flowrate"."B" := "Flowrate"."current in ml/min"."B";
       "Flowrate"."Current Flowrate".mixed := "Flowrate"."current in ml/min".Mixed;
   END_IF;
END_REGION

REGION Network 16: Display flowrate in litre
   RUNG wire#powerrail
      Contact( "Flowrate".Selected.litre )
      wire#w1
      Move(in := "Flowrate"."current in L/min"."A", out1 => "Flowrate"."Current Flowrate"."A")
   END_RUNG
   RUNG wire#w1
      Move(in := "Flowrate"."current in L/min"."B", out1 => "Flowrate"."Current Flowrate"."B")
   END_RUNG
   RUNG wire#w1
      Move(in := "Flowrate"."current in L/min".Mixed, out1 => "Flowrate"."Current Flowrate".mixed)
   END_RUNG
   // the same network as SCL:
   IF "Flowrate".Selected.litre THEN
       "Flowrate"."Current Flowrate"."A" := "Flowrate"."current in L/min"."A";
       "Flowrate"."Current Flowrate"."B" := "Flowrate"."current in L/min"."B";
       "Flowrate"."Current Flowrate".mixed := "Flowrate"."current in L/min".Mixed;
   END_IF;
END_REGION

REGION Network 17: Display flowrate in kg
   RUNG wire#powerrail
      Contact( "Flowrate".Selected.kg )
      wire#w1
      Move(in := "Flowrate"."current in KG/min"."A", out1 => "Flowrate"."Current Flowrate"."A")
   END_RUNG
   RUNG wire#w1
      Move(in := "Flowrate"."current in KG/min"."B", out1 => "Flowrate"."Current Flowrate"."B")
   END_RUNG
   RUNG wire#w1
      Move(in := "Flowrate"."current in KG/min".Mixed, out1 => "Flowrate"."Current Flowrate".mixed)
   END_RUNG
   // the same network as SCL:
   IF "Flowrate".Selected.kg THEN
       "Flowrate"."Current Flowrate"."A" := "Flowrate"."current in KG/min"."A";
       "Flowrate"."Current Flowrate"."B" := "Flowrate"."current in KG/min"."B";
       "Flowrate"."Current Flowrate".mixed := "Flowrate"."current in KG/min".Mixed;
   END_IF;
END_REGION

REGION Network 18: Display flowrate in kg
   RUNG wire#powerrail
      Contact( "Flowrate".Selected.g )
      wire#w1
      Move(in := "Flowrate"."current in g/min"."A", out1 => "Flowrate"."Current Flowrate"."A")
   END_RUNG
   RUNG wire#w1
      Move(in := "Flowrate"."current in g/min"."B", out1 => "Flowrate"."Current Flowrate"."B")
   END_RUNG
   RUNG wire#w1
      Move(in := "Flowrate"."current in g/min".Mixed, out1 => "Flowrate"."Current Flowrate".mixed)
   END_RUNG
   // the same network as SCL:
   IF "Flowrate".Selected.g THEN
       "Flowrate"."Current Flowrate"."A" := "Flowrate"."current in g/min"."A";
       "Flowrate"."Current Flowrate"."B" := "Flowrate"."current in g/min"."B";
       "Flowrate"."Current Flowrate".mixed := "Flowrate"."current in g/min".Mixed;
   END_IF;
END_REGION

REGION Network 19: Flowrate tolerence
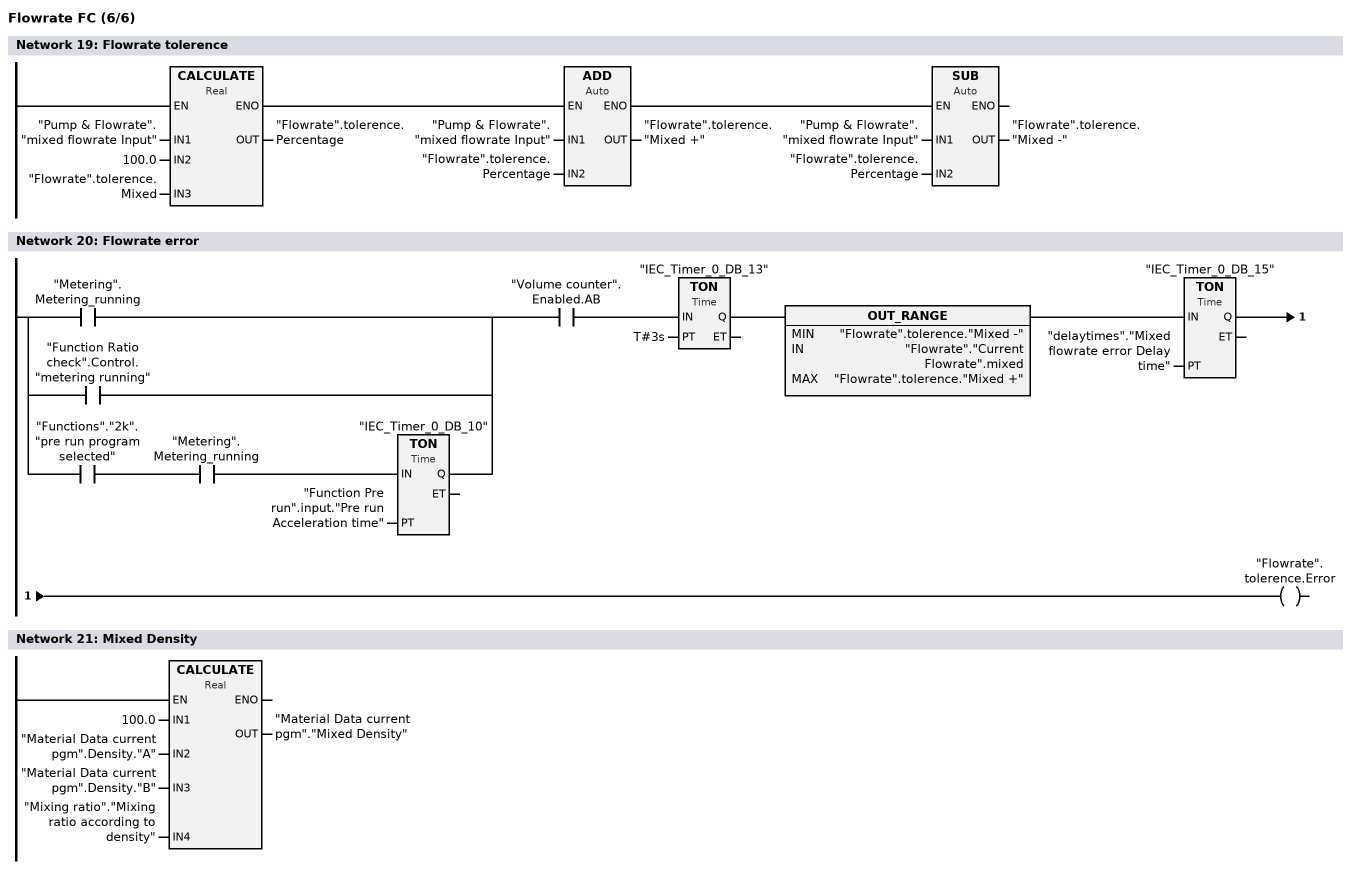
   RUNG wire#powerrail
      { S7_Templates := "SrcType := Real"; S7_Expression := "(IN1/IN2)*IN3" } Calculate(in1 := "Pump & Flowrate"."mixed flowrate Input", in2 := 100.0, in3 := "Flowrate".tolerence.Mixed, out => "Flowrate".tolerence.Percentage)
      Add(in1 := "Pump & Flowrate"."mixed flowrate Input", in2 := "Flowrate".tolerence.Percentage, out => "Flowrate".tolerence."Mixed +")
      Sub(in1 := "Pump & Flowrate"."mixed flowrate Input", in2 := "Flowrate".tolerence.Percentage, out => "Flowrate".tolerence."Mixed -")
   END_RUNG
   // the same network as SCL:
   "Flowrate".tolerence.Percentage := ("Pump & Flowrate"."mixed flowrate Input"/100.0)*"Flowrate".tolerence.Mixed;
   "Flowrate".tolerence."Mixed +" := "Pump & Flowrate"."mixed flowrate Input" + "Flowrate".tolerence.Percentage;
   "Flowrate".tolerence."Mixed -" := "Pump & Flowrate"."mixed flowrate Input" - "Flowrate".tolerence.Percentage;
END_REGION

REGION Network 20: Flowrate error
   "IEC_Timer_0_DB_10".TON(IN := "Functions"."2k"."pre run program selected" AND "Metering".Metering_running,
                           PT := "Function Pre run".input."Pre run Acceleration time");
   "IEC_Timer_0_DB_13".TON(IN := ("Metering".Metering_running OR "Function Ratio check".Control."metering running" OR "IEC_Timer_0_DB_10".Q) AND "Volume counter".Enabled.AB,
                           PT := T#3s);
   "IEC_Timer_0_DB_15".TON(IN := "IEC_Timer_0_DB_13".Q AND (("Flowrate"."Current Flowrate".mixed < "Flowrate".tolerence."Mixed -") OR ("Flowrate"."Current Flowrate".mixed > "Flowrate".tolerence."Mixed +")),
                           PT := "delaytimes"."Mixed flowrate error Delay time");
   "Flowrate".tolerence.Error := "IEC_Timer_0_DB_15".Q;
END_REGION

REGION Network 21: Mixed Density
   RUNG wire#powerrail
      { S7_Templates := "SrcType := Real"; S7_Expression := "(IN2*IN1+IN3*IN4)/(IN1+IN4)" } Calculate(in1 := 100.0, in2 := "Material Data current pgm".Density."A", in3 := "Material Data current pgm".Density."B", in4 := "Mixing ratio"."Mixing ratio according to density", out => "Material Data current pgm"."Mixed Density")
   END_RUNG
   // the same network as SCL:
   "Material Data current pgm"."Mixed Density" := ("Material Data current pgm".Density."A"*100.0+"Material Data current pgm".Density."B"*"Mixing ratio"."Mixing ratio according to density")/(100.0+"Mixing ratio"."Mixing ratio according to density");
END_REGION
END_FUNCTION

FUNCTION "Deaering sequences" : Void   // FC4, LAD
{ S7_Optimized_Access := 'TRUE' }
VERSION : 0.1
// stored: AutoNumber true, IsIECCheckEnabled false, SetENOAutomatically false, UDAEnableTagReadback false
BEGIN

REGION Network 1: Dearing A with valve
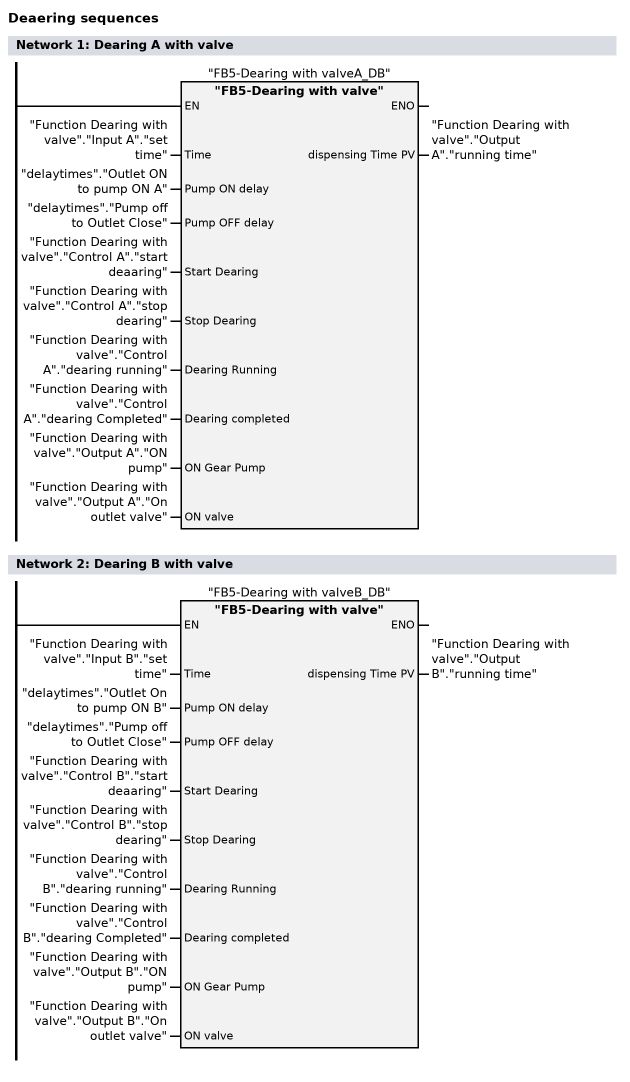
   RUNG wire#powerrail
      "FB5-Dearing with valveA_DB"("Time" := "Function Dearing with valve"."Input A"."set time", "Pump ON delay" := "delaytimes"."Outlet ON to pump ON A", "Pump OFF delay" := "delaytimes"."Pump off to Outlet Close", "Start Dearing" := "Function Dearing with valve"."Control A"."start deaaring", "Stop Dearing" := "Function Dearing with valve"."Control A"."stop dearing", "Dearing Running" := "Function Dearing with valve"."Control A"."dearing running", "Dearing completed" := "Function Dearing with valve"."Control A"."dearing Completed", "ON Gear Pump" := "Function Dearing with valve"."Output A"."ON pump", "ON valve" := "Function Dearing with valve"."Output A"."On outlet valve", "dispensing Time PV" => "Function Dearing with valve"."Output A"."running time")
   END_RUNG
   // the same network as SCL:
   "FB5-Dearing with valveA_DB"("Time" := "Function Dearing with valve"."Input A"."set time",   // "FB5-Dearing with valve"
                           "Pump ON delay" := "delaytimes"."Outlet ON to pump ON A",
                           "Pump OFF delay" := "delaytimes"."Pump off to Outlet Close",
                           "Start Dearing" := "Function Dearing with valve"."Control A"."start deaaring",
                           "Stop Dearing" := "Function Dearing with valve"."Control A"."stop dearing",
                           "Dearing Running" := "Function Dearing with valve"."Control A"."dearing running",
                           "Dearing completed" := "Function Dearing with valve"."Control A"."dearing Completed",
                           "ON Gear Pump" := "Function Dearing with valve"."Output A"."ON pump",
                           "ON valve" := "Function Dearing with valve"."Output A"."On outlet valve",
                           "dispensing Time PV" => "Function Dearing with valve"."Output A"."running time");
END_REGION

REGION Network 2: Dearing B with valve
   RUNG wire#powerrail
      "FB5-Dearing with valveB_DB"("Time" := "Function Dearing with valve"."Input B"."set time", "Pump ON delay" := "delaytimes"."Outlet On to pump ON B", "Pump OFF delay" := "delaytimes"."Pump off to Outlet Close", "Start Dearing" := "Function Dearing with valve"."Control B"."start deaaring", "Stop Dearing" := "Function Dearing with valve"."Control B"."stop dearing", "Dearing Running" := "Function Dearing with valve"."Control B"."dearing running", "Dearing completed" := "Function Dearing with valve"."Control B"."dearing Completed", "ON Gear Pump" := "Function Dearing with valve"."Output B"."ON pump", "ON valve" := "Function Dearing with valve"."Output B"."On outlet valve", "dispensing Time PV" => "Function Dearing with valve"."Output B"."running time")
   END_RUNG
   // the same network as SCL:
   "FB5-Dearing with valveB_DB"("Time" := "Function Dearing with valve"."Input B"."set time",   // "FB5-Dearing with valve"
                           "Pump ON delay" := "delaytimes"."Outlet On to pump ON B",
                           "Pump OFF delay" := "delaytimes"."Pump off to Outlet Close",
                           "Start Dearing" := "Function Dearing with valve"."Control B"."start deaaring",
                           "Stop Dearing" := "Function Dearing with valve"."Control B"."stop dearing",
                           "Dearing Running" := "Function Dearing with valve"."Control B"."dearing running",
                           "Dearing completed" := "Function Dearing with valve"."Control B"."dearing Completed",
                           "ON Gear Pump" := "Function Dearing with valve"."Output B"."ON pump",
                           "ON valve" := "Function Dearing with valve"."Output B"."On outlet valve",
                           "dispensing Time PV" => "Function Dearing with valve"."Output B"."running time");
END_REGION

REGION Network 3: Dearing A without Valve
END_REGION

REGION Network 4: Dearing B without Valve
END_REGION
END_FUNCTION

FUNCTION_BLOCK "FB5-Dearing with valve"   // FB5, LAD
{ S7_Optimized_Access := 'TRUE' }
VERSION : 0.1
// stored: AutoNumber false, IsIECCheckEnabled false, IsRetainMemResEnabled false, MemoryReserve 100, SetENOAutomatically false, UDAEnableTagReadback false
   VAR_INPUT
      "Time" : DInt;
      "Pump ON delay" : DInt;
      "Pump OFF delay" : DInt;
   END_VAR
   VAR_OUTPUT
      "dispensing Time PV" : Int;
   END_VAR
   VAR_IN_OUT
      "Start Dearing" : Bool;
      "Stop Dearing" : Bool;
      "Dearing Running" : Bool;
      "Dearing completed" : Bool;
      "ON Gear Pump" : Bool;
      "ON valve" : Bool;
   END_VAR
   VAR
      "dispensing time done" : Bool;
      "dispensing time in sec" : DInt;
      "timer in sec" : DInt;
      "timer PV in sec" : DInt;
      "timer input" : DInt;
      IEC_Timer_0_Instance { S7_SetPoint := 'True'} : TON_TIME;
      IEC_Timer_0_Instance_1 { S7_SetPoint := 'True'} : TON_TIME;
      IEC_Timer_0_Instance_2 { S7_SetPoint := 'True'} : TON_TIME;
      IEC_Timer_0_Instance_3 { S7_SetPoint := 'True'} : TON_TIME;
   END_VAR
   VAR_TEMP   // added for the SCL form of the ladder/FBD networks
      _w1 : Bool;
   END_VAR
BEGIN

REGION Network 1
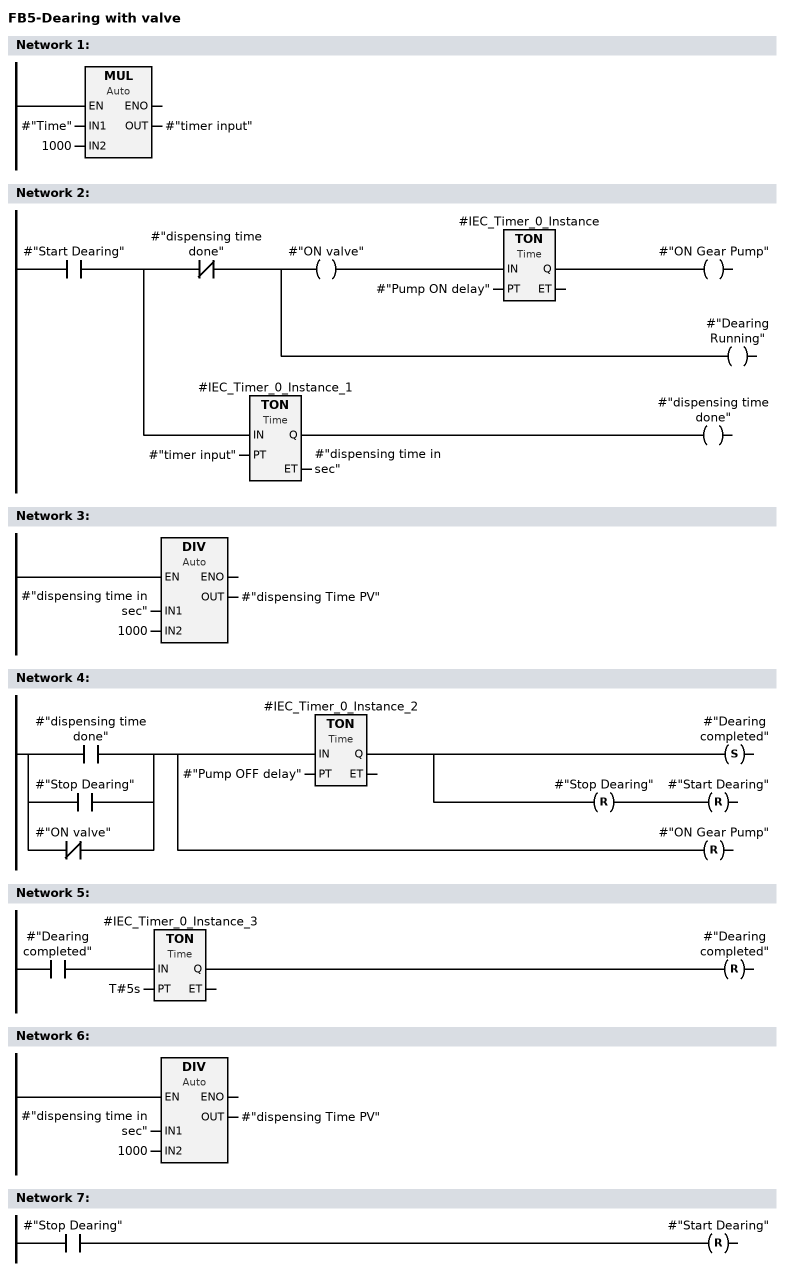
   RUNG wire#powerrail
      Mul(in1 := #"Time", in2 := 1000, out => #"timer input")
   END_RUNG
   // the same network as SCL:
   #"timer input" := #"Time" * 1000;
END_REGION

REGION Network 2
   RUNG wire#powerrail
      Contact( #"Start Dearing" )
      wire#w1
      I_Contact( #"dispensing time done" )
      wire#w2
      Coil( #"ON valve" )
      { S7_Templates := "time_type := Time" } #IEC_Timer_0_Instance.TON(pt := #"Pump ON delay", et =>)
      Coil( #"ON Gear Pump" )
   END_RUNG
   RUNG wire#w2
      Coil( #"Dearing Running" )
   END_RUNG
   RUNG wire#w1
      { S7_Templates := "time_type := Time" } #IEC_Timer_0_Instance_1.TON(pt := #"timer input", et => #"dispensing time in sec")
      Coil( #"dispensing time done" )
   END_RUNG
   // the same network as SCL:
   #"ON valve" := #"Start Dearing" AND NOT #"dispensing time done";
   #IEC_Timer_0_Instance(IN := #"ON valve", PT := #"Pump ON delay");   // TON
   #"ON Gear Pump" := #IEC_Timer_0_Instance.Q;
   #"Dearing Running" := #"ON valve";
   #IEC_Timer_0_Instance_1(IN := #"Start Dearing", PT := #"timer input", ET => #"dispensing time in sec");   // TON
   #"dispensing time done" := #IEC_Timer_0_Instance_1.Q;
END_REGION

REGION Network 3
   RUNG wire#powerrail
      Div(in1 := #"dispensing time in sec", in2 := 1000, out => #"dispensing Time PV")
   END_RUNG
   // the same network as SCL:
   #"dispensing Time PV" := #"dispensing time in sec" / 1000;
END_REGION

REGION Network 4
   RUNG wire#powerrail
      Contact( #"dispensing time done" )
      wire#w1
      { S7_Templates := "time_type := Time" } #IEC_Timer_0_Instance_2.TON(pt := #"Pump OFF delay", et =>)
      wire#w2
      S_Coil( #"Dearing completed" )
   END_RUNG
   RUNG wire#powerrail
      Contact( #"Stop Dearing" )
   END_RUNG wire#w1
   RUNG wire#powerrail
      I_Contact( #"ON valve" )
   END_RUNG wire#w1
   RUNG wire#w2
      R_Coil( #"Stop Dearing" )
      R_Coil( #"Start Dearing" )
   END_RUNG
   RUNG wire#w1
      R_Coil( #"ON Gear Pump" )
   END_RUNG
   // the same network as SCL:
   #_w1 := #"dispensing time done" OR #"Stop Dearing" OR NOT #"ON valve";
   #IEC_Timer_0_Instance_2(IN := #_w1, PT := #"Pump OFF delay");   // TON
   IF #IEC_Timer_0_Instance_2.Q THEN
       #"Dearing completed" := TRUE;
       #"Stop Dearing" := FALSE;
       #"Start Dearing" := FALSE;
   END_IF;
   IF #_w1 THEN #"ON Gear Pump" := FALSE; END_IF;
END_REGION

REGION Network 5
   RUNG wire#powerrail
      Contact( #"Dearing completed" )
      { S7_Templates := "time_type := Time" } #IEC_Timer_0_Instance_3.TON(pt := T#5s, et =>)
      R_Coil( #"Dearing completed" )
   END_RUNG
   // the same network as SCL:
   #IEC_Timer_0_Instance_3(IN := #"Dearing completed", PT := T#5s);   // TON
   IF #IEC_Timer_0_Instance_3.Q THEN #"Dearing completed" := FALSE; END_IF;
END_REGION

REGION Network 6
   RUNG wire#powerrail
      Div(in1 := #"dispensing time in sec", in2 := 1000, out => #"dispensing Time PV")
   END_RUNG
   // the same network as SCL:
   #"dispensing Time PV" := #"dispensing time in sec" / 1000;
END_REGION

REGION Network 7
   RUNG wire#powerrail
      Contact( #"Stop Dearing" )
      R_Coil( #"Start Dearing" )
   END_RUNG
   // the same network as SCL:
   IF #"Stop Dearing" THEN #"Start Dearing" := FALSE; END_IF;
END_REGION
END_FUNCTION_BLOCK

FUNCTION "Flush sequences" : Void   // FC17, LAD
{ S7_Optimized_Access := 'TRUE' }
VERSION : 0.1
// stored: AutoNumber true, IsIECCheckEnabled false, SetENOAutomatically false, UDAEnableTagReadback false
   VAR_TEMP
      temp1 : Bool;
      temp2 : Bool;
   END_VAR
   VAR_TEMP   // added for the SCL form of the ladder/FBD networks
      _w1 : Bool;
      _w2 : Bool;
   END_VAR
BEGIN

REGION Network 1 (SCL)
   IF "Function Flush".Selection = 0 THEN
       "Functions"."flush selection"."Flush A selected" := true;
       "Functions"."flush selection"."Flush B selected" := false;
       "Pump & Flowrate"."Flush Maximum Flowrate" := "Pump & Flowrate".capacity."Pump A";
       "Pump & Flowrate"."Flush minimum Flowrate" := "Pump & Flowrate".capacity."Pump A" * 0.10;
       "Function Flush"."Input A"."set time in sec" := REAL_TO_DINT(("Function Flush"."Input A"."set qty" / "Function Flush"."Input A"."set flowrate") * 60.0);
   ELSE
       "Functions"."flush selection"."Flush A selected" := false;
       "Functions"."flush selection"."Flush B selected" := true;
       "Pump & Flowrate"."Flush Maximum Flowrate" := "Pump & Flowrate".capacity."pump B";
       "Pump & Flowrate"."Flush minimum Flowrate" := "Pump & Flowrate".capacity."pump B" * 0.10;
       "Function Flush"."Input B"."set time in sec" := REAL_TO_DINT(("Function Flush"."Input B"."set qty" / "Function Flush"."Input B"."set flowrate") * 60.0);
   END_IF;
END_REGION

REGION Network 2: Flush A sequences
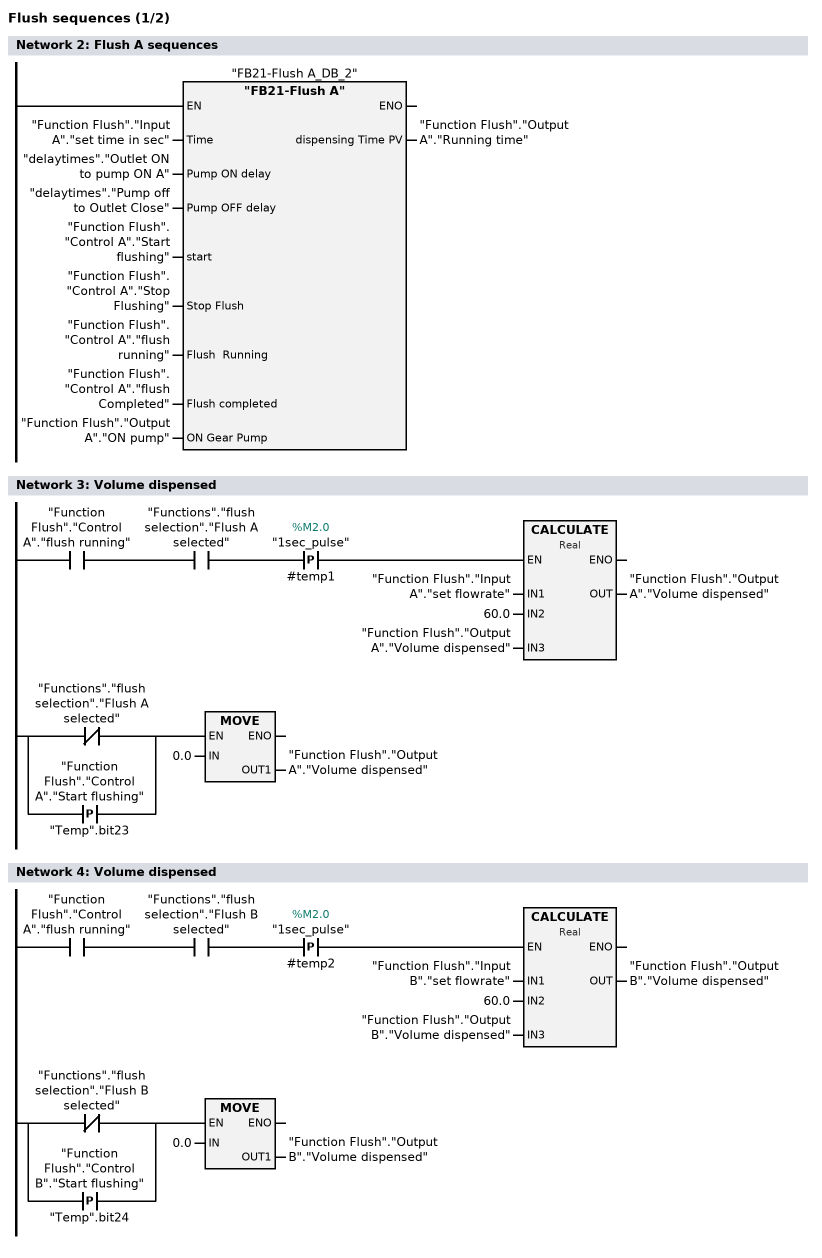
   RUNG wire#powerrail
      "FB21-Flush A_DB_2"("Time" := "Function Flush"."Input A"."set time in sec", "Pump ON delay" := "delaytimes"."Outlet ON to pump ON A", "Pump OFF delay" := "delaytimes"."Pump off to Outlet Close", start := "Function Flush"."Control A"."Start flushing", "Stop Flush" := "Function Flush"."Control A"."Stop Flushing", "Flush  Running" := "Function Flush"."Control A"."flush running", "Flush completed" := "Function Flush"."Control A"."flush Completed", "ON Gear Pump" := "Function Flush"."Output A"."ON pump", "dispensing Time PV" => "Function Flush"."Output A"."Running time")
   END_RUNG
   // the same network as SCL:
   "FB21-Flush A_DB_2"("Time" := "Function Flush"."Input A"."set time in sec",   // "FB21-Flush A"
                       "Pump ON delay" := "delaytimes"."Outlet ON to pump ON A",
                       "Pump OFF delay" := "delaytimes"."Pump off to Outlet Close",
                       start := "Function Flush"."Control A"."Start flushing",
                       "Stop Flush" := "Function Flush"."Control A"."Stop Flushing",
                       "Flush  Running" := "Function Flush"."Control A"."flush running",
                       "Flush completed" := "Function Flush"."Control A"."flush Completed",
                       "ON Gear Pump" := "Function Flush"."Output A"."ON pump",
                       "dispensing Time PV" => "Function Flush"."Output A"."Running time");
END_REGION

REGION Network 3: Volume dispensed
   RUNG wire#powerrail
      Contact( "Function Flush"."Control A"."flush running" )
      Contact( "Functions"."flush selection"."Flush A selected" )
      P_Contact(operand := "1sec_pulse", bit := #temp1)
      { S7_Templates := "SrcType := Real"; S7_Expression := "(IN1/IN2)+IN3" } Calculate(in1 := "Function Flush"."Input A"."set flowrate", in2 := 60.0, in3 := "Function Flush"."Output A"."Volume dispensed", out => "Function Flush"."Output A"."Volume dispensed")
   END_RUNG
   RUNG wire#powerrail
      I_Contact( "Functions"."flush selection"."Flush A selected" )
      wire#w1
      Move(in := 0.0, out1 => "Function Flush"."Output A"."Volume dispensed")
   END_RUNG
   RUNG wire#powerrail
      P_Contact(operand := "Function Flush"."Control A"."Start flushing", bit := "Temp".bit23)
   END_RUNG wire#w1
   // the same network as SCL:
   #_w1 := "Function Flush"."Control A"."flush running" AND "Functions"."flush selection"."Flush A selected" AND "1sec_pulse" AND NOT #temp1;   // rising edge of "1sec_pulse"
   #temp1 := "1sec_pulse";
   IF #_w1 THEN
       "Function Flush"."Output A"."Volume dispensed" := ("Function Flush"."Input A"."set flowrate"/60.0)+"Function Flush"."Output A"."Volume dispensed";
   END_IF;
   #_w2 := "Function Flush"."Control A"."Start flushing" AND NOT "Temp".bit23;   // rising edge of "Function Flush"."Control A"."Start flushing"
   "Temp".bit23 := "Function Flush"."Control A"."Start flushing";
   IF NOT "Functions"."flush selection"."Flush A selected" OR #_w2 THEN
       "Function Flush"."Output A"."Volume dispensed" := 0.0;
   END_IF;
END_REGION

REGION Network 4: Volume dispensed
   RUNG wire#powerrail
      Contact( "Function Flush"."Control A"."flush running" )
      Contact( "Functions"."flush selection"."Flush B selected" )
      P_Contact(operand := "1sec_pulse", bit := #temp2)
      { S7_Templates := "SrcType := Real"; S7_Expression := "(IN1/IN2)+IN3" } Calculate(in1 := "Function Flush"."Input B"."set flowrate", in2 := 60.0, in3 := "Function Flush"."Output B"."Volume dispensed", out => "Function Flush"."Output B"."Volume dispensed")
   END_RUNG
   RUNG wire#powerrail
      I_Contact( "Functions"."flush selection"."Flush B selected" )
      wire#w1
      Move(in := 0.0, out1 => "Function Flush"."Output B"."Volume dispensed")
   END_RUNG
   RUNG wire#powerrail
      P_Contact(operand := "Function Flush"."Control B"."Start flushing", bit := "Temp".bit24)
   END_RUNG wire#w1
   // the same network as SCL:
   #_w1 := "Function Flush"."Control A"."flush running" AND "Functions"."flush selection"."Flush B selected" AND "1sec_pulse" AND NOT #temp2;   // rising edge of "1sec_pulse"
   #temp2 := "1sec_pulse";
   IF #_w1 THEN
       "Function Flush"."Output B"."Volume dispensed" := ("Function Flush"."Input B"."set flowrate"/60.0)+"Function Flush"."Output B"."Volume dispensed";
   END_IF;
   #_w2 := "Function Flush"."Control B"."Start flushing" AND NOT "Temp".bit24;   // rising edge of "Function Flush"."Control B"."Start flushing"
   "Temp".bit24 := "Function Flush"."Control B"."Start flushing";
   IF NOT "Functions"."flush selection"."Flush B selected" OR #_w2 THEN
       "Function Flush"."Output B"."Volume dispensed" := 0.0;
   END_IF;
END_REGION

REGION Network 5: Set Time In hmi
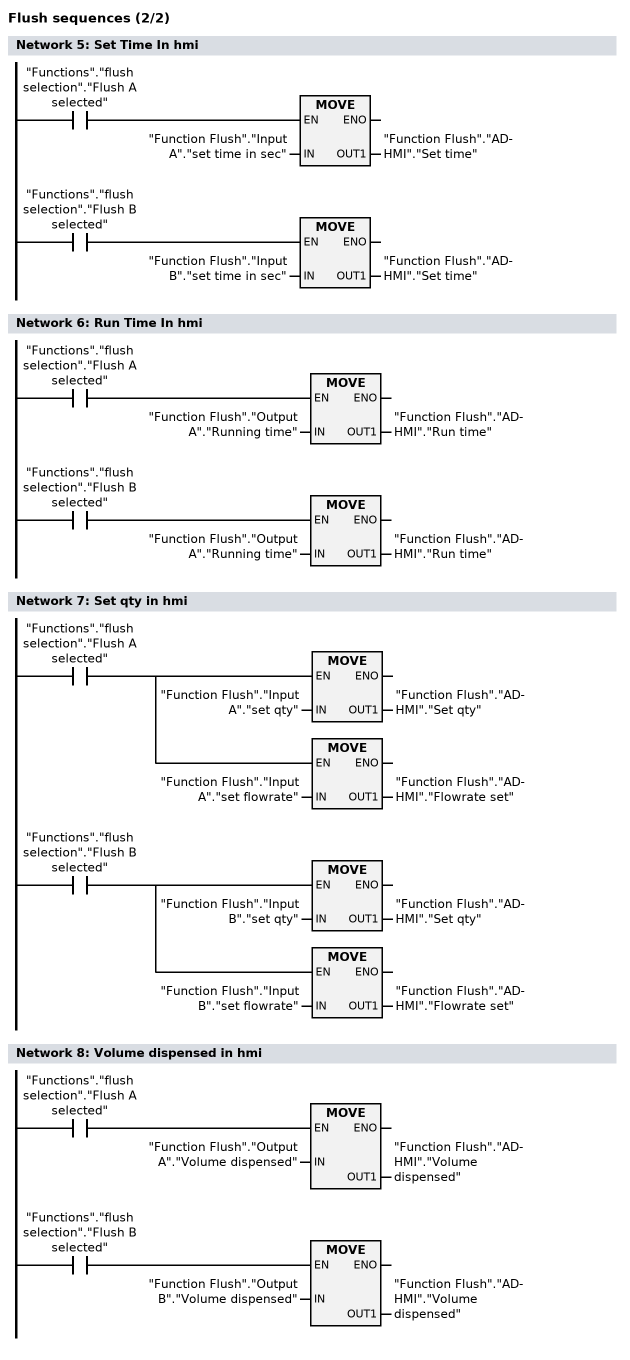
   RUNG wire#powerrail
      Contact( "Functions"."flush selection"."Flush A selected" )
      Move(in := "Function Flush"."Input A"."set time in sec", out1 => "Function Flush"."AD-HMI"."Set time")
   END_RUNG
   RUNG wire#powerrail
      Contact( "Functions"."flush selection"."Flush B selected" )
      Move(in := "Function Flush"."Input B"."set time in sec", out1 => "Function Flush"."AD-HMI"."Set time")
   END_RUNG
   // the same network as SCL:
   IF "Functions"."flush selection"."Flush A selected" THEN
       "Function Flush"."AD-HMI"."Set time" := "Function Flush"."Input A"."set time in sec";
   END_IF;
   IF "Functions"."flush selection"."Flush B selected" THEN
       "Function Flush"."AD-HMI"."Set time" := "Function Flush"."Input B"."set time in sec";
   END_IF;
END_REGION

REGION Network 6: Run Time In hmi
   RUNG wire#powerrail
      Contact( "Functions"."flush selection"."Flush A selected" )
      Move(in := "Function Flush"."Output A"."Running time", out1 => "Function Flush"."AD-HMI"."Run time")
   END_RUNG
   RUNG wire#powerrail
      Contact( "Functions"."flush selection"."Flush B selected" )
      Move(in := "Function Flush"."Output A"."Running time", out1 => "Function Flush"."AD-HMI"."Run time")
   END_RUNG
   // the same network as SCL:
   IF "Functions"."flush selection"."Flush A selected" THEN
       "Function Flush"."AD-HMI"."Run time" := "Function Flush"."Output A"."Running time";
   END_IF;
   IF "Functions"."flush selection"."Flush B selected" THEN
       "Function Flush"."AD-HMI"."Run time" := "Function Flush"."Output A"."Running time";
   END_IF;
END_REGION

REGION Network 7: Set qty in hmi
   RUNG wire#powerrail
      Contact( "Functions"."flush selection"."Flush A selected" )
      wire#w1
      Move(in := "Function Flush"."Input A"."set qty", out1 => "Function Flush"."AD-HMI"."Set qty")
   END_RUNG
   RUNG wire#w1
      Move(in := "Function Flush"."Input A"."set flowrate", out1 => "Function Flush"."AD-HMI"."Flowrate set")
   END_RUNG
   RUNG wire#powerrail
      Contact( "Functions"."flush selection"."Flush B selected" )
      wire#w2
      Move(in := "Function Flush"."Input B"."set qty", out1 => "Function Flush"."AD-HMI"."Set qty")
   END_RUNG
   RUNG wire#w2
      Move(in := "Function Flush"."Input B"."set flowrate", out1 => "Function Flush"."AD-HMI"."Flowrate set")
   END_RUNG
   // the same network as SCL:
   IF "Functions"."flush selection"."Flush A selected" THEN
       "Function Flush"."AD-HMI"."Set qty" := "Function Flush"."Input A"."set qty";
       "Function Flush"."AD-HMI"."Flowrate set" := "Function Flush"."Input A"."set flowrate";
   END_IF;
   IF "Functions"."flush selection"."Flush B selected" THEN
       "Function Flush"."AD-HMI"."Set qty" := "Function Flush"."Input B"."set qty";
       "Function Flush"."AD-HMI"."Flowrate set" := "Function Flush"."Input B"."set flowrate";
   END_IF;
END_REGION

REGION Network 8: Volume dispensed in hmi
   RUNG wire#powerrail
      Contact( "Functions"."flush selection"."Flush A selected" )
      Move(in := "Function Flush"."Output A"."Volume dispensed", out1 => "Function Flush"."AD-HMI"."Volume dispensed")
   END_RUNG
   RUNG wire#powerrail
      Contact( "Functions"."flush selection"."Flush B selected" )
      Move(in := "Function Flush"."Output B"."Volume dispensed", out1 => "Function Flush"."AD-HMI"."Volume dispensed")
   END_RUNG
   // the same network as SCL:
   IF "Functions"."flush selection"."Flush A selected" THEN
       "Function Flush"."AD-HMI"."Volume dispensed" := "Function Flush"."Output A"."Volume dispensed";
   END_IF;
   IF "Functions"."flush selection"."Flush B selected" THEN
       "Function Flush"."AD-HMI"."Volume dispensed" := "Function Flush"."Output B"."Volume dispensed";
   END_IF;
END_REGION
END_FUNCTION

FUNCTION_BLOCK "FB21-Flush A"   // FB21, LAD
{ S7_Optimized_Access := 'TRUE' }
VERSION : 0.1
// stored: AutoNumber false, IsIECCheckEnabled false, IsRetainMemResEnabled false, MemoryReserve 100, SetENOAutomatically false, UDAEnableTagReadback false
   VAR_INPUT
      "Time" : DInt;
      "Pump ON delay" : DInt;
      "Pump OFF delay" : DInt;
   END_VAR
   VAR_OUTPUT
      "dispensing Time PV" : Int;
   END_VAR
   VAR_IN_OUT
      start : Bool;
      "Stop Flush" : Bool;
      "Flush  Running" : Bool;
      "Flush completed" : Bool;
      "ON Gear Pump" : Bool;
   END_VAR
   VAR
      "dispensing time done" : Bool;
      "dispensing time in sec" : DInt;
      "timer input" : DInt;
      IEC_Timer_0_Instance { S7_SetPoint := 'True'} : TON_TIME;
      IEC_Timer_0_Instance_1 { S7_SetPoint := 'True'} : TON_TIME;
      IEC_Timer_0_Instance_2 { S7_SetPoint := 'True'} : TON_TIME;
      IEC_Timer_0_Instance_3 { S7_SetPoint := 'True'} : TON_TIME;
   END_VAR
   VAR_TEMP   // added for the SCL form of the ladder/FBD networks
      _w1 : Bool;
   END_VAR
BEGIN

REGION Network 1
